LIN {X 62.948,Y 54.532,Z 81.721,A 180.000,B 0.000,C 180.000} C_DIS
LIN {X 62.927,Y 54.455,Z 81.718,A 180.000,B 0.000,C 180.000} C_DIS
LIN {X 62.907,Y 54.379,Z 81.716,A 180.000,B 0.000,C 180.000} C_DIS
LIN {X 62.887,Y 54.303,Z 81.713,A 180.000,B 0.000,C 180.000} C_DIS
LIN {X 62.867,Y 54.226,Z 81.710,A 180.000,B 0.000,C 180.000} C_DIS
LIN {X 62.847,Y 54.150,Z 81.707,A 180.000,B 0.000,C 180.000} C_DIS
LIN {X 62.806,Y 53.998,Z 81.702,A 180.000,B 0.000,C 180.000} C_DIS
LIN {X 62.746,Y 53.769,Z 81.693,A 180.000,B 0.000,C 180.000} C_DIS
LIN {X 62.706,Y 53.616,Z 81.688,A 180.000,B 0.000,C 180.000} C_DIS
LIN {X 62.686,Y 53.540,Z 81.685,A 180.000,B 0.000,C 180.000} C_DIS
LIN {X 62.645,Y 53.387,Z 81.680,A 180.000,B 0.000,C 180.000} C_DIS
LIN {X 62.585,Y 53.158,Z 81.671,A 180.000,B 0.000,C 180.000} C_DIS
LIN {X 62.544,Y 53.006,Z 81.666,A 180.000,B 0.000,C 180.000} C_DIS
LIN {X 62.524,Y 52.929,Z 81.663,A 180.000,B 0.000,C 180.000} C_DIS
LIN {X 62.484,Y 52.777,Z 81.658,A 180.000,B 0.000,C 180.000} C_DIS
LIN {X 62.423,Y 52.548,Z 81.649,A 180.000,B 0.000,C 180.000} C_DIS
LIN {X 62.383,Y 52.395,Z 81.644,A 180.000,B 0.000,C 180.000} C_DIS
LIN {X 62.363,Y 52.319,Z 81.641,A 180.000,B 0.000,C 180.000} C_DIS
LIN {X 62.323,Y 52.166,Z 81.636,A 180.000,B 0.000,C 180.000} C_DIS
LIN {X 62.262,Y 51.937,Z 81.627,A 180.000,B 0.000,C 180.000} C_DIS
LIN {X 62.222,Y 51.785,Z 81.622,A 180.000,B 0.000,C 180.000} C_DIS
LIN {X 62.202,Y 51.708,Z 81.619,A 180.000,B 0.000,C 180.000} C_DIS
LIN {X 62.161,Y 51.556,Z 81.614,A 180.000,B 0.000,C 180.000} C_DIS
LIN {X 62.040,Y 51.098,Z 81.597,A 180.000,B 0.000,C 180.000} C_DIS
LIN {X 62.000,Y 50.945,Z 81.592,A 180.000,B 0.000,C 180.000} C_DIS
LIN {X 61.939,Y 50.716,Z 81.583,A 180.000,B 0.000,C 180.000} C_DIS
LIN {X 61.816,Y 50.259,Z 81.567,A 180.000,B 0.000,C 180.000} C_DIS
LIN {X 61.775,Y 50.107,Z 81.561,A 180.000,B 0.000,C 180.000} C_DIS
LIN {X 61.651,Y 49.650,Z 81.545,A 180.000,B 0.000,C 180.000} C_DIS
LIN {X 61.568,Y 49.345,Z 81.534,A 180.000,B 0.000,C 180.000} C_DIS
LIN {X 61.465,Y 48.965,Z 81.520,A 180.000,B 0.000,C 180.000} C_DIS
LIN {X 61.218,Y 48.051,Z 81.487,A 180.000,B 0.000,C 180.000} C_DIS
LIN {X 61.099,Y 47.612,Z 81.471,A 180.000,B 0.000,C 180.000} C_DIS
LIN {X 61.062,Y 47.478,Z 81.466,A 180.000,B 0.000,C 180.000} C_DIS
LIN {X 61.028,Y 47.375,Z 81.462,A 180.000,B 0.000,C 180.000} C_DIS
LIN {X 60.990,Y 47.272,Z 81.458,A 180.000,B 0.000,C 180.000} C_DIS
LIN {X 60.946,Y 47.169,Z 81.455,A 180.000,B 0.000,C 180.000} C_DIS
LIN {X 60.897,Y 47.067,Z 81.451,A 180.000,B 0.000,C 180.000} C_DIS
LIN {X 60.844,Y 46.969,Z 81.447,A 180.000,B 0.000,C 180.000} C_DIS
LIN {X 60.787,Y 46.873,Z 81.443,A 180.000,B 0.000,C 180.000} C_DIS
LIN {X 60.719,Y 46.772,Z 81.439,A 180.000,B 0.000,C 180.000} C_DIS
LIN {X 60.646,Y 46.673,Z 81.434,A 180.000,B 0.000,C 180.000} C_DIS
LIN {X 60.566,Y 46.577,Z 81.430,A 180.000,B 0.000,C 180.000} C_DIS
LIN {X 60.482,Y 46.486,Z 81.426,A 180.000,B 0.000,C 180.000} C_DIS
LIN {X 60.397,Y 46.403,Z 81.421,A 180.000,B 0.000,C 180.000} C_DIS
LIN {X 60.308,Y 46.324,Z 81.417,A 180.000,B 0.000,C 180.000} C_DIS
LIN {X 60.206,Y 46.243,Z 81.413,A 180.000,B 0.000,C 180.000} C_DIS
LIN {X 60.099,Y 46.167,Z 81.408,A 180.000,B 0.000,C 180.000} C_DIS
LIN {X 59.980,Y 46.093,Z 81.403,A 180.000,B 0.000,C 180.000} C_DIS
LIN {X 59.857,Y 46.027,Z 81.398,A 180.000,B 0.000,C 180.000} C_DIS
LIN {X 59.733,Y 45.969,Z 81.394,A 180.000,B 0.000,C 180.000} C_DIS
LIN {X 59.605,Y 45.918,Z 81.389,A 180.000,B 0.000,C 180.000} C_DIS
LIN {X 59.537,Y 45.895,Z 81.386,A 180.000,B 0.000,C 180.000} C_DIS
LIN {X 59.467,Y 45.874,Z 81.384,A 180.000,B 0.000,C 180.000} C_DIS
LIN {X 59.397,Y 45.855,Z 81.381,A 180.000,B 0.000,C 180.000} C_DIS
LIN {X 59.327,Y 45.838,Z 81.379,A 180.000,B 0.000,C 180.000} C_DIS
LIN {X 59.253,Y 45.823,Z 81.376,A 180.000,B 0.000,C 180.000} C_DIS
LIN {X 59.179,Y 45.810,Z 81.373,A 180.000,B 0.000,C 180.000} C_DIS
LIN {X 59.104,Y 45.800,Z 81.371,A 180.000,B 0.000,C 180.000} C_DIS
LIN {X 59.029,Y 45.793,Z 81.368,A 180.000,B 0.000,C 180.000} C_DIS
LIN {X 58.952,Y 45.788,Z 81.366,A 180.000,B 0.000,C 180.000} C_DIS
LIN {X 58.874,Y 45.785,Z 81.363,A 180.000,B 0.000,C 180.000} C_DIS
LIN {X 58.797,Y 45.786,Z 81.360,A 180.000,B 0.000,C 180.000} C_DIS
LIN {X 58.720,Y 45.789,Z 81.357,A 180.000,B 0.000,C 180.000} C_DIS
LIN {X 58.640,Y 45.795,Z 81.355,A 180.000,B 0.000,C 180.000} C_DIS
LIN {X 58.560,Y 45.803,Z 81.352,A 180.000,B 0.000,C 180.000} C_DIS
LIN {X 58.481,Y 45.815,Z 81.349,A 180.000,B 0.000,C 180.000} C_DIS
LIN {X 58.402,Y 45.829,Z 81.346,A 180.000,B 0.000,C 180.000} C_DIS
LIN {X 58.325,Y 45.846,Z 81.343,A 180.000,B 0.000,C 180.000} C_DIS
LIN {X 58.248,Y 45.866,Z 81.341,A 180.000,B 0.000,C 180.000} C_DIS
LIN {X 58.173,Y 45.889,Z 81.338,A 180.000,B 0.000,C 180.000} C_DIS
LIN {X 58.098,Y 45.913,Z 81.335,A 180.000,B 0.000,C 180.000} C_DIS
LIN {X 57.949,Y 45.964,Z 81.330,A 180.000,B 0.000,C 180.000} C_DIS
LIN {X 57.501,Y 46.115,Z 81.313,A 180.000,B 0.000,C 180.000} C_DIS
LIN {X 57.352,Y 46.165,Z 81.308,A 180.000,B 0.000,C 180.000} C_DIS
LIN {X 56.904,Y 46.316,Z 81.291,A 180.000,B 0.000,C 180.000} C_DIS
LIN {X 56.755,Y 46.367,Z 81.286,A 180.000,B 0.000,C 180.000} C_DIS
LIN {X 56.531,Y 46.442,Z 81.277,A 180.000,B 0.000,C 180.000} C_DIS
LIN {X 56.382,Y 46.492,Z 81.272,A 180.000,B 0.000,C 180.000} C_DIS
LIN {X 56.307,Y 46.518,Z 81.269,A 180.000,B 0.000,C 180.000} C_DIS
LIN {X 56.158,Y 46.568,Z 81.264,A 180.000,B 0.000,C 180.000} C_DIS
LIN {X 55.934,Y 46.643,Z 81.255,A 180.000,B 0.000,C 180.000} C_DIS
LIN {X 55.785,Y 46.694,Z 81.250,A 180.000,B 0.000,C 180.000} C_DIS
LIN {X 55.710,Y 46.719,Z 81.247,A 180.000,B 0.000,C 180.000} C_DIS
LIN {X 55.561,Y 46.769,Z 81.242,A 180.000,B 0.000,C 180.000} C_DIS
LIN {X 55.337,Y 46.845,Z 81.233,A 180.000,B 0.000,C 180.000} C_DIS
LIN {X 55.188,Y 46.895,Z 81.228,A 180.000,B 0.000,C 180.000} C_DIS
LIN {X 55.113,Y 46.920,Z 81.225,A 180.000,B 0.000,C 180.000} C_DIS
LIN {X 54.964,Y 46.971,Z 81.220,A 180.000,B 0.000,C 180.000} C_DIS
LIN {X 54.740,Y 47.046,Z 81.211,A 180.000,B 0.000,C 180.000} C_DIS
LIN {X 54.591,Y 47.097,Z 81.206,A 180.000,B 0.000,C 180.000} C_DIS
LIN {X 54.516,Y 47.122,Z 81.203,A 180.000,B 0.000,C 180.000} C_DIS
LIN {X 54.367,Y 47.172,Z 81.198,A 180.000,B 0.000,C 180.000} C_DIS
LIN {X 54.143,Y 47.248,Z 81.189,A 180.000,B 0.000,C 180.000} C_DIS
LIN {X 53.994,Y 47.298,Z 81.184,A 180.000,B 0.000,C 180.000} C_DIS
LIN {X 53.845,Y 47.348,Z 81.179,A 180.000,B 0.000,C 180.000} C_DIS
LIN {X 53.695,Y 47.399,Z 81.173,A 180.000,B 0.000,C 180.000} C_DIS
LIN {X 53.546,Y 47.449,Z 81.168,A 180.000,B 0.000,C 180.000} C_DIS
LIN {X 53.397,Y 47.499,Z 81.163,A 180.000,B 0.000,C 180.000} C_DIS
LIN {X 53.322,Y 47.524,Z 81.160,A 180.000,B 0.000,C 180.000} C_DIS
LIN {X 53.248,Y 47.550,Z 81.158,A 180.000,B 0.000,C 180.000} C_DIS
LIN {X 53.173,Y 47.575,Z 81.155,A 180.000,B 0.000,C 180.000} C_DIS
LIN {X 53.098,Y 47.600,Z 81.153,A 180.000,B 0.000,C 180.000} C_DIS
LIN {X 53.024,Y 47.625,Z 81.150,A 180.000,B 0.000,C 180.000} C_DIS
LIN {X 52.949,Y 47.650,Z 81.147,A 180.000,B 0.000,C 180.000} C_DIS
LIN {X 52.875,Y 47.675,Z 81.145,A 180.000,B 0.000,C 180.000} C_DIS
LIN {X 52.725,Y 47.726,Z 81.140,A 180.000,B 0.000,C 180.000} C_DIS
LIN {X 52.576,Y 47.776,Z 81.135,A 180.000,B 0.000,C 180.000} C_DIS
LIN {X 52.427,Y 47.827,Z 81.130,A 180.000,B 0.000,C 180.000} C_DIS
LIN {X 52.278,Y 47.877,Z 81.126,A 180.000,B 0.000,C 180.000} C_DIS
LIN {X 52.128,Y 47.927,Z 81.121,A 180.000,B 0.000,C 180.000} C_DIS
LIN {X 51.979,Y 47.978,Z 81.116,A 180.000,B 0.000,C 180.000} C_DIS
LIN {X 51.830,Y 48.028,Z 81.112,A 180.000,B 0.000,C 180.000} C_DIS
LIN {X 51.681,Y 48.078,Z 81.107,A 180.000,B 0.000,C 180.000} C_DIS
LIN {X 51.531,Y 48.129,Z 81.103,A 180.000,B 0.000,C 180.000} C_DIS
LIN {X 51.382,Y 48.179,Z 81.099,A 180.000,B 0.000,C 180.000} C_DIS
LIN {X 51.233,Y 48.229,Z 81.094,A 180.000,B 0.000,C 180.000} C_DIS
LIN {X 51.084,Y 48.280,Z 81.090,A 180.000,B 0.000,C 180.000} C_DIS
LIN {X 50.935,Y 48.330,Z 81.086,A 180.000,B 0.000,C 180.000} C_DIS
LIN {X 50.785,Y 48.380,Z 81.082,A 180.000,B 0.000,C 180.000} C_DIS
LIN {X 50.636,Y 48.431,Z 81.078,A 180.000,B 0.000,C 180.000} C_DIS
LIN {X 50.487,Y 48.481,Z 81.074,A 180.000,B 0.000,C 180.000} C_DIS
LIN {X 50.338,Y 48.531,Z 81.071,A 180.000,B 0.000,C 180.000} C_DIS
LIN {X 50.188,Y 48.582,Z 81.067,A 180.000,B 0.000,C 180.000} C_DIS
LIN {X 50.039,Y 48.632,Z 81.063,A 180.000,B 0.000,C 180.000} C_DIS
LIN {X 49.890,Y 48.682,Z 81.060,A 180.000,B 0.000,C 180.000} C_DIS
LIN {X 49.741,Y 48.733,Z 81.057,A 180.000,B 0.000,C 180.000} C_DIS
LIN {X 49.591,Y 48.783,Z 81.053,A 180.000,B 0.000,C 180.000} C_DIS
LIN {X 49.442,Y 48.833,Z 81.050,A 180.000,B 0.000,C 180.000} C_DIS
LIN {X 49.293,Y 48.884,Z 81.047,A 180.000,B 0.000,C 180.000} C_DIS
LIN {X 49.144,Y 48.934,Z 81.044,A 180.000,B 0.000,C 180.000} C_DIS
LIN {X 48.994,Y 48.984,Z 81.041,A 180.000,B 0.000,C 180.000} C_DIS
LIN {X 48.845,Y 49.035,Z 81.038,A 180.000,B 0.000,C 180.000} C_DIS
LIN {X 48.696,Y 49.085,Z 81.035,A 180.000,B 0.000,C 180.000} C_DIS
LIN {X 48.547,Y 49.135,Z 81.032,A 180.000,B 0.000,C 180.000} C_DIS
LIN {X 48.398,Y 49.186,Z 81.030,A 180.000,B 0.000,C 180.000} C_DIS
LIN {X 48.248,Y 49.236,Z 81.027,A 180.000,B 0.000,C 180.000} C_DIS
LIN {X 47.950,Y 49.337,Z 81.023,A 180.000,B 0.000,C 180.000} C_DIS
LIN {X 47.651,Y 49.438,Z 81.019,A 180.000,B 0.000,C 180.000} C_DIS
LIN {X 47.353,Y 49.538,Z 81.015,A 180.000,B 0.000,C 180.000} C_DIS
LIN {X 47.054,Y 49.639,Z 81.011,A 180.000,B 0.000,C 180.000} C_DIS
LIN {X 46.756,Y 49.740,Z 81.008,A 180.000,B 0.000,C 180.000} C_DIS
LIN {X 46.457,Y 49.840,Z 81.006,A 180.000,B 0.000,C 180.000} C_DIS
LIN {X 46.159,Y 49.941,Z 81.004,A 180.000,B 0.000,C 180.000} C_DIS
LIN {X 46.085,Y 49.969,Z 81.003,A 180.000,B 0.000,C 180.000} C_DIS
LIN {X 46.013,Y 49.999,Z 81.003,A 180.000,B 0.000,C 180.000} C_DIS
LIN {X 45.941,Y 50.032,Z 81.002,A 180.000,B 0.000,C 180.000} C_DIS
LIN {X 45.870,Y 50.066,Z 81.002,A 180.000,B 0.000,C 180.000} C_DIS
LIN {X 45.800,Y 50.103,Z 81.002,A 180.000,B 0.000,C 180.000} C_DIS
LIN {X 45.732,Y 50.142,Z 81.001,A 180.000,B 0.000,C 180.000} C_DIS
LIN {X 45.665,Y 50.183,Z 81.001,A 180.000,B 0.000,C 180.000} C_DIS
LIN {X 45.599,Y 50.226,Z 81.001,A 180.000,B 0.000,C 180.000} C_DIS
LIN {X 45.534,Y 50.271,Z 81.001,A 180.000,B 0.000,C 180.000} C_DIS
LIN {X 45.471,Y 50.318,Z 81.000,A 180.000,B 0.000,C 180.000} C_DIS
LIN {X 45.410,Y 50.367,Z 81.000,A 180.000,B 0.000,C 180.000} C_DIS
LIN {X 45.350,Y 50.418,Z 81.000,A 180.000,B 0.000,C 180.000} C_DIS
LIN {X 45.250,Y 50.511,Z 81.000,A 180.000,B 0.000,C 180.000} C_DIS
LIN {X 45.156,Y 50.609,Z 81.000,A 180.000,B 0.000,C 180.000} C_DIS
; Cutting Move Starts
LIN {X 45.053,Y 50.728,Z 81.000,A 180.000,B 0.000,C 180.000} C_DIS
LIN {X 45.017,Y 50.774,Z 81.000,A 180.000,B 0.000,C 180.000} C_DIS
LIN {X 44.952,Y 50.863,Z 81.000,A 180.000,B 0.000,C 180.000} C_DIS
LIN {X 44.892,Y 50.953,Z 81.000,A 180.000,B 0.000,C 180.000} C_DIS
LIN {X 44.874,Y 50.981,Z 81.000,A 180.000,B 0.000,C 180.000} C_DIS
LIN {X 44.788,Y 51.131,Z 81.000,A 180.000,B 0.000,C 180.000} C_DIS
LIN {X 44.703,Y 51.310,Z 81.000,A 180.000,B 0.000,C 180.000} C_DIS
LIN {X 44.696,Y 51.328,Z 81.000,A 180.000,B 0.000,C 180.000} C_DIS
LIN {X 44.634,Y 51.489,Z 81.000,A 180.000,B 0.000,C 180.000} C_DIS
LIN {X 44.581,Y 51.668,Z 81.000,A 180.000,B 0.000,C 180.000} C_DIS
LIN {X 44.541,Y 51.847,Z 81.000,A 180.000,B 0.000,C 180.000} C_DIS
LIN {X 44.517,Y 52.012,Z 81.000,A 180.000,B 0.000,C 180.000} C_DIS
LIN {X 44.515,Y 52.025,Z 81.000,A 180.000,B 0.000,C 180.000} C_DIS
LIN {X 44.503,Y 52.204,Z 81.000,A 180.000,B 0.000,C 180.000} C_DIS
LIN {X 44.502,Y 52.383,Z 81.000,A 180.000,B 0.000,C 180.000} C_DIS
LIN {X 44.515,Y 52.562,Z 81.000,A 180.000,B 0.000,C 180.000} C_DIS
LIN {X 44.517,Y 52.579,Z 81.000,A 180.000,B 0.000,C 180.000} C_DIS
LIN {X 44.541,Y 52.740,Z 81.000,A 180.000,B 0.000,C 180.000} C_DIS
LIN {X 44.580,Y 52.919,Z 81.000,A 180.000,B 0.000,C 180.000} C_DIS
LIN {X 44.633,Y 53.098,Z 81.000,A 180.000,B 0.000,C 180.000} C_DIS
LIN {X 51.026,Y 72.048,Z 81.000,A 180.000,B 0.000,C 180.000} C_DIS
LIN {X 51.094,Y 72.226,Z 81.000,A 180.000,B 0.000,C 180.000} C_DIS
LIN {X 51.131,Y 72.310,Z 81.000,A 180.000,B 0.000,C 180.000} C_DIS
LIN {X 51.179,Y 72.405,Z 81.000,A 180.000,B 0.000,C 180.000} C_DIS
LIN {X 51.282,Y 72.584,Z 81.000,A 180.000,B 0.000,C 180.000} C_DIS
LIN {X 51.310,Y 72.628,Z 81.000,A 180.000,B 0.000,C 180.000} C_DIS
LIN {X 51.406,Y 72.763,Z 81.000,A 180.000,B 0.000,C 180.000} C_DIS
LIN {X 51.489,Y 72.865,Z 81.000,A 180.000,B 0.000,C 180.000} C_DIS
LIN {X 51.556,Y 72.941,Z 81.000,A 180.000,B 0.000,C 180.000} C_DIS
LIN {X 51.668,Y 73.055,Z 81.000,A 180.000,B 0.000,C 180.000} C_DIS
LIN {X 51.739,Y 73.120,Z 81.000,A 180.000,B 0.000,C 180.000} C_DIS
LIN {X 51.847,Y 73.210,Z 81.000,A 180.000,B 0.000,C 180.000} C_DIS
LIN {X 51.967,Y 73.299,Z 81.000,A 180.000,B 0.000,C 180.000} C_DIS
LIN {X 52.025,Y 73.338,Z 81.000,A 180.000,B 0.000,C 180.000} C_DIS
LIN {X 52.204,Y 73.445,Z 81.000,A 180.000,B 0.000,C 180.000} C_DIS
LIN {X 52.267,Y 73.478,Z 81.000,A 180.000,B 0.000,C 180.000} C_DIS
LIN {X 52.383,Y 73.533,Z 81.000,A 180.000,B 0.000,C 180.000} C_DIS
LIN {X 52.562,Y 73.604,Z 81.000,A 180.000,B 0.000,C 180.000} C_DIS
LIN {X 52.730,Y 73.656,Z 81.000,A 180.000,B 0.000,C 180.000} C_DIS
LIN {X 52.740,Y 73.659,Z 81.000,A 180.000,B 0.000,C 180.000} C_DIS
LIN {X 52.919,Y 73.701,Z 81.000,A 180.000,B 0.000,C 180.000} C_DIS
LIN {X 53.009,Y 73.716,Z 81.000,A 180.000,B 0.000,C 180.000} C_DIS
LIN {X 53.098,Y 73.729,Z 81.000,A 180.000,B 0.000,C 180.000} C_DIS
LIN {X 53.187,Y 73.738,Z 81.000,A 180.000,B 0.000,C 180.000} C_DIS
LIN {X 53.277,Y 73.743,Z 81.000,A 180.000,B 0.000,C 180.000} C_DIS
LIN {X 53.366,Y 73.746,Z 81.000,A 180.000,B 0.000,C 180.000} C_DIS
LIN {X 53.455,Y 73.745,Z 81.000,A 180.000,B 0.000,C 180.000} C_DIS
LIN {X 53.545,Y 73.742,Z 81.000,A 180.000,B 0.000,C 180.000} C_DIS
LIN {X 53.634,Y 73.735,Z 81.000,A 180.000,B 0.000,C 180.000} C_DIS
LIN {X 53.724,Y 73.724,Z 81.000,A 180.000,B 0.000,C 180.000} C_DIS
LIN {X 53.813,Y 73.711,Z 81.000,A 180.000,B 0.000,C 180.000} C_DIS
LIN {X 53.902,Y 73.694,Z 81.000,A 180.000,B 0.000,C 180.000} C_DIS
LIN {X 53.992,Y 73.674,Z 81.000,A 180.000,B 0.000,C 180.000} C_DIS
LIN {X 54.057,Y 73.656,Z 81.000,A 180.000,B 0.000,C 180.000} C_DIS
LIN {X 54.171,Y 73.622,Z 81.000,A 180.000,B 0.000,C 180.000} C_DIS
LIN {X 54.349,Y 73.562,Z 81.000,A 180.000,B 0.000,C 180.000} C_DIS
LIN {X 66.506,Y 69.461,Z 81.000,A 180.000,B 0.000,C 180.000} C_DIS
LIN {X 66.684,Y 69.401,Z 81.000,A 180.000,B 0.000,C 180.000} C_DIS
LIN {X 66.777,Y 69.366,Z 81.000,A 180.000,B 0.000,C 180.000} C_DIS
LIN {X 66.863,Y 69.330,Z 81.000,A 180.000,B 0.000,C 180.000} C_DIS
LIN {X 66.953,Y 69.288,Z 81.000,A 180.000,B 0.000,C 180.000} C_DIS
LIN {X 67.042,Y 69.242,Z 81.000,A 180.000,B 0.000,C 180.000} C_DIS
LIN {X 67.137,Y 69.187,Z 81.000,A 180.000,B 0.000,C 180.000} C_DIS
LIN {X 67.221,Y 69.135,Z 81.000,A 180.000,B 0.000,C 180.000} C_DIS
LIN {X 67.309,Y 69.074,Z 81.000,A 180.000,B 0.000,C 180.000} C_DIS
LIN {X 67.396,Y 69.008,Z 81.000,A 180.000,B 0.000,C 180.000} C_DIS
LIN {X 67.399,Y 69.006,Z 81.000,A 180.000,B 0.000,C 180.000} C_DIS
LIN {X 67.489,Y 68.932,Z 81.000,A 180.000,B 0.000,C 180.000} C_DIS
LIN {X 67.578,Y 68.850,Z 81.000,A 180.000,B 0.000,C 180.000} C_DIS
LIN {X 67.600,Y 68.830,Z 81.000,A 180.000,B 0.000,C 180.000} C_DIS
LIN {X 67.682,Y 68.745,Z 81.000,A 180.000,B 0.000,C 180.000} C_DIS
LIN {X 67.757,Y 68.661,Z 81.000,A 180.000,B 0.000,C 180.000} C_DIS
LIN {X 67.765,Y 68.651,Z 81.000,A 180.000,B 0.000,C 180.000} C_DIS
LIN {X 67.837,Y 68.562,Z 81.000,A 180.000,B 0.000,C 180.000} C_DIS
LIN {X 67.902,Y 68.472,Z 81.000,A 180.000,B 0.000,C 180.000} C_DIS
LIN {X 67.936,Y 68.422,Z 81.000,A 180.000,B 0.000,C 180.000} C_DIS
LIN {X 68.015,Y 68.293,Z 81.000,A 180.000,B 0.000,C 180.000} C_DIS
LIN {X 68.109,Y 68.115,Z 81.000,A 180.000,B 0.000,C 180.000} C_DIS
LIN {X 68.115,Y 68.103,Z 81.000,A 180.000,B 0.000,C 180.000} C_DIS
LIN {X 68.186,Y 67.936,Z 81.000,A 180.000,B 0.000,C 180.000} C_DIS
LIN {X 68.246,Y 67.757,Z 81.000,A 180.000,B 0.000,C 180.000} C_DIS
LIN {X 68.292,Y 67.578,Z 81.000,A 180.000,B 0.000,C 180.000} C_DIS
LIN {X 68.293,Y 67.573,Z 81.000,A 180.000,B 0.000,C 180.000} C_DIS
LIN {X 68.325,Y 67.399,Z 81.000,A 180.000,B 0.000,C 180.000} C_DIS
LIN {X 68.344,Y 67.221,Z 81.000,A 180.000,B 0.000,C 180.000} C_DIS
LIN {X 68.350,Y 67.042,Z 81.000,A 180.000,B 0.000,C 180.000} C_DIS
LIN {X 68.343,Y 66.863,Z 81.000,A 180.000,B 0.000,C 180.000} C_DIS
LIN {X 68.324,Y 66.684,Z 81.000,A 180.000,B 0.000,C 180.000} C_DIS
LIN {X 68.293,Y 66.515,Z 81.000,A 180.000,B 0.000,C 180.000} C_DIS
LIN {X 68.291,Y 66.506,Z 81.000,A 180.000,B 0.000,C 180.000} C_DIS
LIN {X 68.245,Y 66.327,Z 81.000,A 180.000,B 0.000,C 180.000} C_DIS
LIN {X 68.186,Y 66.148,Z 81.000,A 180.000,B 0.000,C 180.000} C_DIS
LIN {X 61.854,Y 47.377,Z 81.000,A 180.000,B 0.000,C 180.000} C_DIS
LIN {X 61.791,Y 47.198,Z 81.000,A 180.000,B 0.000,C 180.000} C_DIS
LIN {X 61.715,Y 47.020,Z 81.000,A 180.000,B 0.000,C 180.000} C_DIS
LIN {X 61.679,Y 46.947,Z 81.000,A 180.000,B 0.000,C 180.000} C_DIS
LIN {X 61.621,Y 46.841,Z 81.000,A 180.000,B 0.000,C 180.000} C_DIS
LIN {X 61.507,Y 46.662,Z 81.000,A 180.000,B 0.000,C 180.000} C_DIS
LIN {X 61.500,Y 46.653,Z 81.000,A 180.000,B 0.000,C 180.000} C_DIS
LIN {X 61.370,Y 46.483,Z 81.000,A 180.000,B 0.000,C 180.000} C_DIS
LIN {X 61.321,Y 46.428,Z 81.000,A 180.000,B 0.000,C 180.000} C_DIS
LIN {X 61.204,Y 46.305,Z 81.000,A 180.000,B 0.000,C 180.000} C_DIS
LIN {X 61.143,Y 46.247,Z 81.000,A 180.000,B 0.000,C 180.000} C_DIS
LIN {X 60.999,Y 46.126,Z 81.000,A 180.000,B 0.000,C 180.000} C_DIS
LIN {X 60.964,Y 46.098,Z 81.000,A 180.000,B 0.000,C 180.000} C_DIS
LIN {X 60.785,Y 45.975,Z 81.000,A 180.000,B 0.000,C 180.000} C_DIS
LIN {X 60.739,Y 45.947,Z 81.000,A 180.000,B 0.000,C 180.000} C_DIS
LIN {X 60.606,Y 45.873,Z 81.000,A 180.000,B 0.000,C 180.000} C_DIS
LIN {X 60.427,Y 45.789,Z 81.000,A 180.000,B 0.000,C 180.000} C_DIS
LIN {X 60.376,Y 45.768,Z 81.000,A 180.000,B 0.000,C 180.000} C_DIS
LIN {X 60.249,Y 45.722,Z 81.000,A 180.000,B 0.000,C 180.000} C_DIS
LIN {X 60.070,Y 45.670,Z 81.000,A 180.000,B 0.000,C 180.000} C_DIS
LIN {X 59.891,Y 45.631,Z 81.000,A 180.000,B 0.000,C 180.000} C_DIS
LIN {X 59.802,Y 45.617,Z 81.000,A 180.000,B 0.000,C 180.000} C_DIS
LIN {X 59.712,Y 45.606,Z 81.000,A 180.000,B 0.000,C 180.000} C_DIS
LIN {X 59.623,Y 45.599,Z 81.000,A 180.000,B 0.000,C 180.000} C_DIS
LIN {X 59.534,Y 45.595,Z 81.000,A 180.000,B 0.000,C 180.000} C_DIS
LIN {X 59.444,Y 45.593,Z 81.000,A 180.000,B 0.000,C 180.000} C_DIS
LIN {X 59.355,Y 45.595,Z 81.000,A 180.000,B 0.000,C 180.000} C_DIS
LIN {X 59.265,Y 45.601,Z 81.000,A 180.000,B 0.000,C 180.000} C_DIS
LIN {X 59.176,Y 45.609,Z 81.000,A 180.000,B 0.000,C 180.000} C_DIS
LIN {X 59.087,Y 45.621,Z 81.000,A 180.000,B 0.000,C 180.000} C_DIS
LIN {X 58.997,Y 45.636,Z 81.000,A 180.000,B 0.000,C 180.000} C_DIS
LIN {X 58.908,Y 45.654,Z 81.000,A 180.000,B 0.000,C 180.000} C_DIS
LIN {X 58.819,Y 45.676,Z 81.000,A 180.000,B 0.000,C 180.000} C_DIS
LIN {X 58.729,Y 45.702,Z 81.000,A 180.000,B 0.000,C 180.000} C_DIS
LIN {X 58.640,Y 45.731,Z 81.000,A 180.000,B 0.000,C 180.000} C_DIS
LIN {X 46.305,Y 49.892,Z 81.000,A 180.000,B 0.000,C 180.000} C_DIS
LIN {X 46.126,Y 49.954,Z 81.000,A 180.000,B 0.000,C 180.000} C_DIS
LIN {X 46.036,Y 49.989,Z 81.000,A 180.000,B 0.000,C 180.000} C_DIS
LIN {X 45.947,Y 50.028,Z 81.000,A 180.000,B 0.000,C 180.000} C_DIS
LIN {X 45.884,Y 50.059,Z 81.000,A 180.000,B 0.000,C 180.000} C_DIS
LIN {X 45.826,Y 50.089,Z 81.000,A 180.000,B 0.000,C 180.000} C_DIS
LIN {X 45.768,Y 50.120,Z 81.000,A 180.000,B 0.000,C 180.000} C_DIS
LIN {X 45.679,Y 50.173,Z 81.000,A 180.000,B 0.000,C 180.000} C_DIS
LIN {X 45.590,Y 50.232,Z 81.000,A 180.000,B 0.000,C 180.000} C_DIS
LIN {X 45.581,Y 50.238,Z 81.000,A 180.000,B 0.000,C 180.000} C_DIS
LIN {X 45.496,Y 50.299,Z 81.000,A 180.000,B 0.000,C 180.000} C_DIS
LIN {X 45.411,Y 50.366,Z 81.000,A 180.000,B 0.000,C 180.000} C_DIS
LIN {X 45.352,Y 50.416,Z 81.000,A 180.000,B 0.000,C 180.000} C_DIS
LIN {X 45.232,Y 50.529,Z 81.000,A 180.000,B 0.000,C 180.000} C_DIS
LIN {X 45.168,Y 50.595,Z 81.000,A 180.000,B 0.000,C 180.000} C_DIS
LIN {X 45.156,Y 50.609,Z 81.000,A 180.000,B 0.000,C 180.000} C_DIS
; Link Move Starts
LIN {X 45.061,Y 50.718,Z 81.000,A 180.000,B 0.000,C 180.000} C_DIS
LIN {X 44.974,Y 50.832,Z 81.000,A 180.000,B 0.000,C 180.000} C_DIS
LIN {X 44.894,Y 50.948,Z 81.000,A 180.000,B 0.000,C 180.000} C_DIS
LIN {X 44.822,Y 51.068,Z 80.999,A 180.000,B 0.000,C 180.000} C_DIS
LIN {X 44.761,Y 51.182,Z 80.999,A 180.000,B 0.000,C 180.000} C_DIS
LIN {X 44.706,Y 51.299,Z 80.998,A 180.000,B 0.000,C 180.000} C_DIS
LIN {X 44.657,Y 51.418,Z 80.998,A 180.000,B 0.000,C 180.000} C_DIS
LIN {X 44.614,Y 51.539,Z 80.997,A 180.000,B 0.000,C 180.000} C_DIS
LIN {X 44.553,Y 51.760,Z 80.996,A 180.000,B 0.000,C 180.000} C_DIS
LIN {X 44.527,Y 51.892,Z 80.995,A 180.000,B 0.000,C 180.000} C_DIS
LIN {X 44.507,Y 52.025,Z 80.994,A 180.000,B 0.000,C 180.000} C_DIS
LIN {X 44.490,Y 52.238,Z 80.992,A 180.000,B 0.000,C 180.000} C_DIS
LIN {X 44.491,Y 52.450,Z 80.990,A 180.000,B 0.000,C 180.000} C_DIS
LIN {X 44.512,Y 52.682,Z 80.988,A 180.000,B 0.000,C 180.000} C_DIS
LIN {X 44.531,Y 52.799,Z 80.986,A 180.000,B 0.000,C 180.000} C_DIS
LIN {X 44.555,Y 52.914,Z 80.985,A 180.000,B 0.000,C 180.000} C_DIS
LIN {X 44.611,Y 53.117,Z 80.983,A 180.000,B 0.000,C 180.000} C_DIS
LIN {X 44.705,Y 53.413,Z 80.978,A 180.000,B 0.000,C 180.000} C_DIS
LIN {X 44.799,Y 53.714,Z 80.974,A 180.000,B 0.000,C 180.000} C_DIS
LIN {X 44.892,Y 54.014,Z 80.969,A 180.000,B 0.000,C 180.000} C_DIS
LIN {X 44.939,Y 54.165,Z 80.966,A 180.000,B 0.000,C 180.000} C_DIS
LIN {X 44.985,Y 54.316,Z 80.964,A 180.000,B 0.000,C 180.000} C_DIS
LIN {X 45.031,Y 54.466,Z 80.961,A 180.000,B 0.000,C 180.000} C_DIS
LIN {X 45.078,Y 54.617,Z 80.958,A 180.000,B 0.000,C 180.000} C_DIS
LIN {X 45.124,Y 54.768,Z 80.955,A 180.000,B 0.000,C 180.000} C_DIS
LIN {X 45.169,Y 54.918,Z 80.952,A 180.000,B 0.000,C 180.000} C_DIS
LIN {X 45.215,Y 55.069,Z 80.949,A 180.000,B 0.000,C 180.000} C_DIS
LIN {X 45.261,Y 55.220,Z 80.945,A 180.000,B 0.000,C 180.000} C_DIS
LIN {X 45.306,Y 55.371,Z 80.942,A 180.000,B 0.000,C 180.000} C_DIS
LIN {X 45.352,Y 55.522,Z 80.939,A 180.000,B 0.000,C 180.000} C_DIS
LIN {X 45.397,Y 55.673,Z 80.935,A 180.000,B 0.000,C 180.000} C_DIS
LIN {X 45.442,Y 55.824,Z 80.931,A 180.000,B 0.000,C 180.000} C_DIS
LIN {X 45.487,Y 55.975,Z 80.928,A 180.000,B 0.000,C 180.000} C_DIS
LIN {X 45.532,Y 56.126,Z 80.924,A 180.000,B 0.000,C 180.000} C_DIS
LIN {X 45.576,Y 56.277,Z 80.920,A 180.000,B 0.000,C 180.000} C_DIS
LIN {X 45.621,Y 56.428,Z 80.916,A 180.000,B 0.000,C 180.000} C_DIS
LIN {X 45.666,Y 56.579,Z 80.912,A 180.000,B 0.000,C 180.000} C_DIS
LIN {X 45.710,Y 56.731,Z 80.908,A 180.000,B 0.000,C 180.000} C_DIS
LIN {X 45.754,Y 56.882,Z 80.904,A 180.000,B 0.000,C 180.000} C_DIS
LIN {X 45.798,Y 57.033,Z 80.899,A 180.000,B 0.000,C 180.000} C_DIS
LIN {X 45.842,Y 57.185,Z 80.895,A 180.000,B 0.000,C 180.000} C_DIS
LIN {X 45.886,Y 57.336,Z 80.891,A 180.000,B 0.000,C 180.000} C_DIS
LIN {X 45.930,Y 57.487,Z 80.886,A 180.000,B 0.000,C 180.000} C_DIS
LIN {X 45.974,Y 57.639,Z 80.882,A 180.000,B 0.000,C 180.000} C_DIS
LIN {X 46.018,Y 57.790,Z 80.877,A 180.000,B 0.000,C 180.000} C_DIS
LIN {X 46.061,Y 57.942,Z 80.872,A 180.000,B 0.000,C 180.000} C_DIS
LIN {X 46.105,Y 58.093,Z 80.868,A 180.000,B 0.000,C 180.000} C_DIS
LIN {X 46.148,Y 58.245,Z 80.863,A 180.000,B 0.000,C 180.000} C_DIS
LIN {X 46.191,Y 58.397,Z 80.858,A 180.000,B 0.000,C 180.000} C_DIS
LIN {X 46.234,Y 58.548,Z 80.853,A 180.000,B 0.000,C 180.000} C_DIS
LIN {X 46.256,Y 58.624,Z 80.850,A 180.000,B 0.000,C 180.000} C_DIS
LIN {X 46.277,Y 58.700,Z 80.848,A 180.000,B 0.000,C 180.000} C_DIS
LIN {X 46.299,Y 58.776,Z 80.845,A 180.000,B 0.000,C 180.000} C_DIS
LIN {X 46.320,Y 58.852,Z 80.843,A 180.000,B 0.000,C 180.000} C_DIS
LIN {X 46.342,Y 58.928,Z 80.840,A 180.000,B 0.000,C 180.000} C_DIS
LIN {X 46.363,Y 59.004,Z 80.838,A 180.000,B 0.000,C 180.000} C_DIS
LIN {X 46.385,Y 59.079,Z 80.835,A 180.000,B 0.000,C 180.000} C_DIS
LIN {X 46.406,Y 59.155,Z 80.832,A 180.000,B 0.000,C 180.000} C_DIS
LIN {X 46.427,Y 59.231,Z 80.830,A 180.000,B 0.000,C 180.000} C_DIS
LIN {X 46.449,Y 59.307,Z 80.827,A 180.000,B 0.000,C 180.000} C_DIS
LIN {X 46.470,Y 59.383,Z 80.824,A 180.000,B 0.000,C 180.000} C_DIS
LIN {X 46.491,Y 59.459,Z 80.822,A 180.000,B 0.000,C 180.000} C_DIS
LIN {X 46.513,Y 59.535,Z 80.819,A 180.000,B 0.000,C 180.000} C_DIS
LIN {X 46.534,Y 59.611,Z 80.816,A 180.000,B 0.000,C 180.000} C_DIS
LIN {X 46.555,Y 59.687,Z 80.814,A 180.000,B 0.000,C 180.000} C_DIS
LIN {X 46.597,Y 59.839,Z 80.808,A 180.000,B 0.000,C 180.000} C_DIS
LIN {X 46.619,Y 59.915,Z 80.805,A 180.000,B 0.000,C 180.000} C_DIS
LIN {X 46.640,Y 59.991,Z 80.803,A 180.000,B 0.000,C 180.000} C_DIS
LIN {X 46.661,Y 60.067,Z 80.800,A 180.000,B 0.000,C 180.000} C_DIS
LIN {X 46.682,Y 60.143,Z 80.797,A 180.000,B 0.000,C 180.000} C_DIS
LIN {X 46.703,Y 60.219,Z 80.794,A 180.000,B 0.000,C 180.000} C_DIS
LIN {X 46.725,Y 60.295,Z 80.792,A 180.000,B 0.000,C 180.000} C_DIS
LIN {X 46.746,Y 60.370,Z 80.789,A 180.000,B 0.000,C 180.000} C_DIS
LIN {X 46.767,Y 60.446,Z 80.786,A 180.000,B 0.000,C 180.000} C_DIS
LIN {X 46.788,Y 60.522,Z 80.783,A 180.000,B 0.000,C 180.000} C_DIS
LIN {X 46.809,Y 60.598,Z 80.781,A 180.000,B 0.000,C 180.000} C_DIS
LIN {X 46.830,Y 60.674,Z 80.778,A 180.000,B 0.000,C 180.000} C_DIS
LIN {X 46.852,Y 60.750,Z 80.775,A 180.000,B 0.000,C 180.000} C_DIS
LIN {X 46.873,Y 60.826,Z 80.772,A 180.000,B 0.000,C 180.000} C_DIS
LIN {X 46.894,Y 60.902,Z 80.770,A 180.000,B 0.000,C 180.000} C_DIS
LIN {X 46.915,Y 60.978,Z 80.767,A 180.000,B 0.000,C 180.000} C_DIS
LIN {X 46.936,Y 61.054,Z 80.764,A 180.000,B 0.000,C 180.000} C_DIS
LIN {X 46.958,Y 61.130,Z 80.761,A 180.000,B 0.000,C 180.000} C_DIS
LIN {X 46.979,Y 61.206,Z 80.759,A 180.000,B 0.000,C 180.000} C_DIS
LIN {X 47.000,Y 61.282,Z 80.756,A 180.000,B 0.000,C 180.000} C_DIS
LIN {X 47.021,Y 61.358,Z 80.753,A 180.000,B 0.000,C 180.000} C_DIS
LIN {X 47.042,Y 61.434,Z 80.750,A 180.000,B 0.000,C 180.000} C_DIS
LIN {X 47.063,Y 61.510,Z 80.748,A 180.000,B 0.000,C 180.000} C_DIS
LIN {X 47.085,Y 61.586,Z 80.745,A 180.000,B 0.000,C 180.000} C_DIS
LIN {X 47.106,Y 61.662,Z 80.742,A 180.000,B 0.000,C 180.000} C_DIS
LIN {X 47.149,Y 61.814,Z 80.737,A 180.000,B 0.000,C 180.000} C_DIS
LIN {X 47.170,Y 61.890,Z 80.734,A 180.000,B 0.000,C 180.000} C_DIS
LIN {X 47.213,Y 62.041,Z 80.728,A 180.000,B 0.000,C 180.000} C_DIS
LIN {X 47.277,Y 62.269,Z 80.720,A 180.000,B 0.000,C 180.000} C_DIS
LIN {X 47.320,Y 62.421,Z 80.714,A 180.000,B 0.000,C 180.000} C_DIS
LIN {X 47.341,Y 62.497,Z 80.712,A 180.000,B 0.000,C 180.000} C_DIS
LIN {X 47.384,Y 62.648,Z 80.706,A 180.000,B 0.000,C 180.000} C_DIS
LIN {X 47.448,Y 62.876,Z 80.698,A 180.000,B 0.000,C 180.000} C_DIS
LIN {X 47.491,Y 63.028,Z 80.692,A 180.000,B 0.000,C 180.000} C_DIS
LIN {X 47.512,Y 63.104,Z 80.690,A 180.000,B 0.000,C 180.000} C_DIS
LIN {X 47.555,Y 63.256,Z 80.684,A 180.000,B 0.000,C 180.000} C_DIS
LIN {X 47.619,Y 63.483,Z 80.676,A 180.000,B 0.000,C 180.000} C_DIS
LIN {X 47.662,Y 63.635,Z 80.670,A 180.000,B 0.000,C 180.000} C_DIS
LIN {X 47.683,Y 63.711,Z 80.668,A 180.000,B 0.000,C 180.000} C_DIS
LIN {X 47.726,Y 63.863,Z 80.662,A 180.000,B 0.000,C 180.000} C_DIS
LIN {X 47.790,Y 64.091,Z 80.654,A 180.000,B 0.000,C 180.000} C_DIS
LIN {X 47.833,Y 64.242,Z 80.648,A 180.000,B 0.000,C 180.000} C_DIS
LIN {X 47.854,Y 64.318,Z 80.646,A 180.000,B 0.000,C 180.000} C_DIS
LIN {X 47.897,Y 64.470,Z 80.640,A 180.000,B 0.000,C 180.000} C_DIS
LIN {X 48.025,Y 64.925,Z 80.624,A 180.000,B 0.000,C 180.000} C_DIS
LIN {X 48.068,Y 65.077,Z 80.618,A 180.000,B 0.000,C 180.000} C_DIS
LIN {X 48.196,Y 65.533,Z 80.602,A 180.000,B 0.000,C 180.000} C_DIS
LIN {X 48.261,Y 65.760,Z 80.593,A 180.000,B 0.000,C 180.000} C_DIS
LIN {X 48.303,Y 65.912,Z 80.588,A 180.000,B 0.000,C 180.000} C_DIS
LIN {X 48.432,Y 66.367,Z 80.571,A 180.000,B 0.000,C 180.000} C_DIS
LIN {X 48.474,Y 66.519,Z 80.566,A 180.000,B 0.000,C 180.000} C_DIS
LIN {X 48.667,Y 67.202,Z 80.541,A 180.000,B 0.000,C 180.000} C_DIS
LIN {X 49.052,Y 68.568,Z 80.491,A 180.000,B 0.000,C 180.000} C_DIS
LIN {X 49.243,Y 69.247,Z 80.467,A 180.000,B 0.000,C 180.000} C_DIS
LIN {X 49.244,Y 69.251,Z 80.467,A 180.000,B 0.000,C 180.000} C_DIS
LIN {X 49.949,Y 71.341,Z 80.390,A 180.000,B 0.000,C 180.000} C_DIS
LIN {X 50.100,Y 71.788,Z 80.373,A 180.000,B 0.000,C 180.000} C_DIS
LIN {X 50.151,Y 71.938,Z 80.368,A 180.000,B 0.000,C 180.000} C_DIS
LIN {X 50.251,Y 72.236,Z 80.357,A 180.000,B 0.000,C 180.000} C_DIS
LIN {X 50.276,Y 72.311,Z 80.354,A 180.000,B 0.000,C 180.000} C_DIS
LIN {X 50.303,Y 72.385,Z 80.351,A 180.000,B 0.000,C 180.000} C_DIS
LIN {X 50.332,Y 72.458,Z 80.348,A 180.000,B 0.000,C 180.000} C_DIS
LIN {X 50.364,Y 72.530,Z 80.346,A 180.000,B 0.000,C 180.000} C_DIS
LIN {X 50.397,Y 72.602,Z 80.343,A 180.000,B 0.000,C 180.000} C_DIS
LIN {X 50.433,Y 72.672,Z 80.340,A 180.000,B 0.000,C 180.000} C_DIS
LIN {X 50.471,Y 72.741,Z 80.337,A 180.000,B 0.000,C 180.000} C_DIS
LIN {X 50.511,Y 72.808,Z 80.335,A 180.000,B 0.000,C 180.000} C_DIS
LIN {X 50.553,Y 72.875,Z 80.332,A 180.000,B 0.000,C 180.000} C_DIS
LIN {X 50.598,Y 72.940,Z 80.329,A 180.000,B 0.000,C 180.000} C_DIS
LIN {X 50.644,Y 73.004,Z 80.326,A 180.000,B 0.000,C 180.000} C_DIS
LIN {X 50.692,Y 73.066,Z 80.324,A 180.000,B 0.000,C 180.000} C_DIS
LIN {X 50.743,Y 73.126,Z 80.321,A 180.000,B 0.000,C 180.000} C_DIS
LIN {X 50.795,Y 73.185,Z 80.318,A 180.000,B 0.000,C 180.000} C_DIS
LIN {X 50.849,Y 73.243,Z 80.315,A 180.000,B 0.000,C 180.000} C_DIS
LIN {X 50.905,Y 73.298,Z 80.313,A 180.000,B 0.000,C 180.000} C_DIS
LIN {X 50.962,Y 73.352,Z 80.310,A 180.000,B 0.000,C 180.000} C_DIS
LIN {X 51.021,Y 73.404,Z 80.307,A 180.000,B 0.000,C 180.000} C_DIS
LIN {X 51.082,Y 73.454,Z 80.304,A 180.000,B 0.000,C 180.000} C_DIS
LIN {X 51.144,Y 73.502,Z 80.302,A 180.000,B 0.000,C 180.000} C_DIS
LIN {X 51.208,Y 73.549,Z 80.299,A 180.000,B 0.000,C 180.000} C_DIS
LIN {X 51.274,Y 73.593,Z 80.296,A 180.000,B 0.000,C 180.000} C_DIS
LIN {X 51.340,Y 73.635,Z 80.293,A 180.000,B 0.000,C 180.000} C_DIS
LIN {X 51.408,Y 73.675,Z 80.291,A 180.000,B 0.000,C 180.000} C_DIS
LIN {X 51.477,Y 73.712,Z 80.288,A 180.000,B 0.000,C 180.000} C_DIS
LIN {X 51.547,Y 73.748,Z 80.285,A 180.000,B 0.000,C 180.000} C_DIS
LIN {X 51.619,Y 73.781,Z 80.282,A 180.000,B 0.000,C 180.000} C_DIS
LIN {X 51.691,Y 73.812,Z 80.280,A 180.000,B 0.000,C 180.000} C_DIS
LIN {X 51.764,Y 73.841,Z 80.277,A 180.000,B 0.000,C 180.000} C_DIS
LIN {X 51.839,Y 73.868,Z 80.274,A 180.000,B 0.000,C 180.000} C_DIS
LIN {X 51.914,Y 73.892,Z 80.271,A 180.000,B 0.000,C 180.000} C_DIS
LIN {X 51.989,Y 73.913,Z 80.269,A 180.000,B 0.000,C 180.000} C_DIS
LIN {X 52.066,Y 73.933,Z 80.266,A 180.000,B 0.000,C 180.000} C_DIS
LIN {X 52.143,Y 73.950,Z 80.263,A 180.000,B 0.000,C 180.000} C_DIS
LIN {X 52.220,Y 73.964,Z 80.260,A 180.000,B 0.000,C 180.000} C_DIS
LIN {X 52.298,Y 73.976,Z 80.258,A 180.000,B 0.000,C 180.000} C_DIS
LIN {X 52.376,Y 73.986,Z 80.255,A 180.000,B 0.000,C 180.000} C_DIS
LIN {X 52.454,Y 73.993,Z 80.252,A 180.000,B 0.000,C 180.000} C_DIS
LIN {X 52.533,Y 73.998,Z 80.250,A 180.000,B 0.000,C 180.000} C_DIS
LIN {X 52.612,Y 74.000,Z 80.247,A 180.000,B 0.000,C 180.000} C_DIS
LIN {X 52.691,Y 74.000,Z 80.244,A 180.000,B 0.000,C 180.000} C_DIS
LIN {X 52.769,Y 73.997,Z 80.241,A 180.000,B 0.000,C 180.000} C_DIS
LIN {X 52.848,Y 73.991,Z 80.239,A 180.000,B 0.000,C 180.000} C_DIS
LIN {X 52.926,Y 73.984,Z 80.236,A 180.000,B 0.000,C 180.000} C_DIS
LIN {X 53.004,Y 73.973,Z 80.233,A 180.000,B 0.000,C 180.000} C_DIS
LIN {X 53.082,Y 73.961,Z 80.230,A 180.000,B 0.000,C 180.000} C_DIS
LIN {X 53.159,Y 73.946,Z 80.228,A 180.000,B 0.000,C 180.000} C_DIS
LIN {X 53.236,Y 73.928,Z 80.225,A 180.000,B 0.000,C 180.000} C_DIS
LIN {X 53.312,Y 73.908,Z 80.222,A 180.000,B 0.000,C 180.000} C_DIS
LIN {X 53.388,Y 73.886,Z 80.219,A 180.000,B 0.000,C 180.000} C_DIS
LIN {X 53.463,Y 73.861,Z 80.217,A 180.000,B 0.000,C 180.000} C_DIS
LIN {X 53.612,Y 73.811,Z 80.211,A 180.000,B 0.000,C 180.000} C_DIS
LIN {X 53.836,Y 73.735,Z 80.203,A 180.000,B 0.000,C 180.000} C_DIS
LIN {X 53.985,Y 73.685,Z 80.197,A 180.000,B 0.000,C 180.000} C_DIS
LIN {X 54.060,Y 73.660,Z 80.195,A 180.000,B 0.000,C 180.000} C_DIS
LIN {X 54.209,Y 73.610,Z 80.189,A 180.000,B 0.000,C 180.000} C_DIS
LIN {X 54.358,Y 73.559,Z 80.184,A 180.000,B 0.000,C 180.000} C_DIS
LIN {X 54.507,Y 73.509,Z 80.178,A 180.000,B 0.000,C 180.000} C_DIS
LIN {X 54.657,Y 73.459,Z 80.173,A 180.000,B 0.000,C 180.000} C_DIS
LIN {X 54.806,Y 73.408,Z 80.168,A 180.000,B 0.000,C 180.000} C_DIS
LIN {X 54.881,Y 73.383,Z 80.165,A 180.000,B 0.000,C 180.000} C_DIS
LIN {X 54.955,Y 73.358,Z 80.162,A 180.000,B 0.000,C 180.000} C_DIS
LIN {X 55.030,Y 73.333,Z 80.160,A 180.000,B 0.000,C 180.000} C_DIS
LIN {X 55.104,Y 73.308,Z 80.157,A 180.000,B 0.000,C 180.000} C_DIS
LIN {X 55.179,Y 73.282,Z 80.155,A 180.000,B 0.000,C 180.000} C_DIS
LIN {X 55.254,Y 73.257,Z 80.152,A 180.000,B 0.000,C 180.000} C_DIS
LIN {X 55.328,Y 73.232,Z 80.150,A 180.000,B 0.000,C 180.000} C_DIS
LIN {X 55.403,Y 73.207,Z 80.147,A 180.000,B 0.000,C 180.000} C_DIS
LIN {X 55.552,Y 73.156,Z 80.142,A 180.000,B 0.000,C 180.000} C_DIS
LIN {X 55.701,Y 73.106,Z 80.137,A 180.000,B 0.000,C 180.000} C_DIS
LIN {X 55.851,Y 73.056,Z 80.132,A 180.000,B 0.000,C 180.000} C_DIS
LIN {X 56.000,Y 73.005,Z 80.128,A 180.000,B 0.000,C 180.000} C_DIS
LIN {X 56.149,Y 72.955,Z 80.123,A 180.000,B 0.000,C 180.000} C_DIS
LIN {X 56.298,Y 72.905,Z 80.118,A 180.000,B 0.000,C 180.000} C_DIS
LIN {X 56.448,Y 72.854,Z 80.114,A 180.000,B 0.000,C 180.000} C_DIS
LIN {X 56.597,Y 72.804,Z 80.109,A 180.000,B 0.000,C 180.000} C_DIS
LIN {X 56.746,Y 72.754,Z 80.105,A 180.000,B 0.000,C 180.000} C_DIS
LIN {X 56.895,Y 72.703,Z 80.100,A 180.000,B 0.000,C 180.000} C_DIS
LIN {X 57.044,Y 72.653,Z 80.096,A 180.000,B 0.000,C 180.000} C_DIS
LIN {X 57.194,Y 72.603,Z 80.092,A 180.000,B 0.000,C 180.000} C_DIS
LIN {X 57.343,Y 72.552,Z 80.088,A 180.000,B 0.000,C 180.000} C_DIS
LIN {X 57.492,Y 72.502,Z 80.084,A 180.000,B 0.000,C 180.000} C_DIS
LIN {X 57.641,Y 72.452,Z 80.080,A 180.000,B 0.000,C 180.000} C_DIS
LIN {X 57.791,Y 72.401,Z 80.076,A 180.000,B 0.000,C 180.000} C_DIS
LIN {X 57.940,Y 72.351,Z 80.072,A 180.000,B 0.000,C 180.000} C_DIS
LIN {X 58.089,Y 72.301,Z 80.069,A 180.000,B 0.000,C 180.000} C_DIS
LIN {X 58.238,Y 72.250,Z 80.065,A 180.000,B 0.000,C 180.000} C_DIS
LIN {X 58.388,Y 72.200,Z 80.061,A 180.000,B 0.000,C 180.000} C_DIS
LIN {X 58.537,Y 72.150,Z 80.058,A 180.000,B 0.000,C 180.000} C_DIS
LIN {X 58.686,Y 72.099,Z 80.055,A 180.000,B 0.000,C 180.000} C_DIS
LIN {X 58.835,Y 72.049,Z 80.051,A 180.000,B 0.000,C 180.000} C_DIS
LIN {X 58.985,Y 71.999,Z 80.048,A 180.000,B 0.000,C 180.000} C_DIS
LIN {X 59.134,Y 71.948,Z 80.045,A 180.000,B 0.000,C 180.000} C_DIS
LIN {X 59.283,Y 71.898,Z 80.042,A 180.000,B 0.000,C 180.000} C_DIS
LIN {X 59.432,Y 71.848,Z 80.039,A 180.000,B 0.000,C 180.000} C_DIS
LIN {X 59.581,Y 71.797,Z 80.036,A 180.000,B 0.000,C 180.000} C_DIS
LIN {X 59.731,Y 71.747,Z 80.034,A 180.000,B 0.000,C 180.000} C_DIS
LIN {X 59.880,Y 71.696,Z 80.031,A 180.000,B 0.000,C 180.000} C_DIS
LIN {X 60.029,Y 71.646,Z 80.028,A 180.000,B 0.000,C 180.000} C_DIS
LIN {X 60.328,Y 71.545,Z 80.024,A 180.000,B 0.000,C 180.000} C_DIS
LIN {X 60.626,Y 71.445,Z 80.019,A 180.000,B 0.000,C 180.000} C_DIS
LIN {X 60.925,Y 71.344,Z 80.015,A 180.000,B 0.000,C 180.000} C_DIS
LIN {X 61.223,Y 71.243,Z 80.012,A 180.000,B 0.000,C 180.000} C_DIS
LIN {X 61.522,Y 71.143,Z 80.009,A 180.000,B 0.000,C 180.000} C_DIS
LIN {X 61.820,Y 71.042,Z 80.006,A 180.000,B 0.000,C 180.000} C_DIS
LIN {X 62.118,Y 70.941,Z 80.004,A 180.000,B 0.000,C 180.000} C_DIS
LIN {X 62.417,Y 70.841,Z 80.002,A 180.000,B 0.000,C 180.000} C_DIS
LIN {X 62.715,Y 70.740,Z 80.001,A 180.000,B 0.000,C 180.000} C_DIS
LIN {X 63.014,Y 70.639,Z 80.000,A 180.000,B 0.000,C 180.000} C_DIS
LIN {X 63.312,Y 70.539,Z 80.000,A 180.000,B 0.000,C 180.000} C_DIS
LIN {X 63.340,Y 70.529,Z 80.000,A 180.000,B 0.000,C 180.000} C_DIS
; Cutting Move Starts
LIN {X 67.936,Y 68.979,Z 80.000,A 180.000,B 0.000,C 180.000} C_DIS
LIN {X 68.115,Y 68.917,Z 80.000,A 180.000,B 0.000,C 180.000} C_DIS
LIN {X 68.204,Y 68.882,Z 80.000,A 180.000,B 0.000,C 180.000} C_DIS
LIN {X 68.293,Y 68.842,Z 80.000,A 180.000,B 0.000,C 180.000} C_DIS
LIN {X 68.320,Y 68.830,Z 80.000,A 180.000,B 0.000,C 180.000} C_DIS
LIN {X 68.396,Y 68.792,Z 80.000,A 180.000,B 0.000,C 180.000} C_DIS
LIN {X 68.472,Y 68.750,Z 80.000,A 180.000,B 0.000,C 180.000} C_DIS
LIN {X 68.553,Y 68.703,Z 80.000,A 180.000,B 0.000,C 180.000} C_DIS
LIN {X 68.633,Y 68.651,Z 80.000,A 180.000,B 0.000,C 180.000} C_DIS
LIN {X 68.651,Y 68.639,Z 80.000,A 180.000,B 0.000,C 180.000} C_DIS
LIN {X 68.740,Y 68.575,Z 80.000,A 180.000,B 0.000,C 180.000} C_DIS
LIN {X 68.830,Y 68.504,Z 80.000,A 180.000,B 0.000,C 180.000} C_DIS
LIN {X 68.868,Y 68.472,Z 80.000,A 180.000,B 0.000,C 180.000} C_DIS
LIN {X 68.938,Y 68.409,Z 80.000,A 180.000,B 0.000,C 180.000} C_DIS
LIN {X 69.008,Y 68.342,Z 80.000,A 180.000,B 0.000,C 180.000} C_DIS
LIN {X 69.056,Y 68.293,Z 80.000,A 180.000,B 0.000,C 180.000} C_DIS
LIN {X 69.124,Y 68.218,Z 80.000,A 180.000,B 0.000,C 180.000} C_DIS
LIN {X 69.187,Y 68.142,Z 80.000,A 180.000,B 0.000,C 180.000} C_DIS
LIN {X 69.209,Y 68.115,Z 80.000,A 180.000,B 0.000,C 180.000} C_DIS
LIN {X 69.276,Y 68.025,Z 80.000,A 180.000,B 0.000,C 180.000} C_DIS
LIN {X 69.337,Y 67.936,Z 80.000,A 180.000,B 0.000,C 180.000} C_DIS
LIN {X 69.366,Y 67.890,Z 80.000,A 180.000,B 0.000,C 180.000} C_DIS
LIN {X 69.442,Y 67.757,Z 80.000,A 180.000,B 0.000,C 180.000} C_DIS
LIN {X 69.529,Y 67.578,Z 80.000,A 180.000,B 0.000,C 180.000} C_DIS
LIN {X 69.545,Y 67.542,Z 80.000,A 180.000,B 0.000,C 180.000} C_DIS
LIN {X 69.600,Y 67.399,Z 80.000,A 180.000,B 0.000,C 180.000} C_DIS
LIN {X 69.655,Y 67.221,Z 80.000,A 180.000,B 0.000,C 180.000} C_DIS
LIN {X 69.695,Y 67.042,Z 80.000,A 180.000,B 0.000,C 180.000} C_DIS
LIN {X 69.723,Y 66.863,Z 80.000,A 180.000,B 0.000,C 180.000} C_DIS
LIN {X 69.724,Y 66.856,Z 80.000,A 180.000,B 0.000,C 180.000} C_DIS
LIN {X 69.737,Y 66.684,Z 80.000,A 180.000,B 0.000,C 180.000} C_DIS
LIN {X 69.738,Y 66.506,Z 80.000,A 180.000,B 0.000,C 180.000} C_DIS
LIN {X 69.727,Y 66.327,Z 80.000,A 180.000,B 0.000,C 180.000} C_DIS
LIN {X 69.724,Y 66.295,Z 80.000,A 180.000,B 0.000,C 180.000} C_DIS
LIN {X 69.703,Y 66.148,Z 80.000,A 180.000,B 0.000,C 180.000} C_DIS
LIN {X 69.665,Y 65.969,Z 80.000,A 180.000,B 0.000,C 180.000} C_DIS
LIN {X 69.613,Y 65.791,Z 80.000,A 180.000,B 0.000,C 180.000} C_DIS
LIN {X 69.553,Y 65.612,Z 80.000,A 180.000,B 0.000,C 180.000} C_DIS
LIN {X 63.220,Y 46.841,Z 80.000,A 180.000,B 0.000,C 180.000} C_DIS
LIN {X 63.154,Y 46.662,Z 80.000,A 180.000,B 0.000,C 180.000} C_DIS
LIN {X 63.109,Y 46.562,Z 80.000,A 180.000,B 0.000,C 180.000} C_DIS
LIN {X 63.071,Y 46.483,Z 80.000,A 180.000,B 0.000,C 180.000} C_DIS
LIN {X 62.969,Y 46.305,Z 80.000,A 180.000,B 0.000,C 180.000} C_DIS
LIN {X 62.930,Y 46.244,Z 80.000,A 180.000,B 0.000,C 180.000} C_DIS
LIN {X 62.847,Y 46.126,Z 80.000,A 180.000,B 0.000,C 180.000} C_DIS
LIN {X 62.751,Y 46.006,Z 80.000,A 180.000,B 0.000,C 180.000} C_DIS
LIN {X 62.700,Y 45.947,Z 80.000,A 180.000,B 0.000,C 180.000} C_DIS
LIN {X 62.573,Y 45.816,Z 80.000,A 180.000,B 0.000,C 180.000} C_DIS
LIN {X 62.521,Y 45.768,Z 80.000,A 180.000,B 0.000,C 180.000} C_DIS
LIN {X 62.394,Y 45.661,Z 80.000,A 180.000,B 0.000,C 180.000} C_DIS
LIN {X 62.298,Y 45.590,Z 80.000,A 180.000,B 0.000,C 180.000} C_DIS
LIN {X 62.215,Y 45.533,Z 80.000,A 180.000,B 0.000,C 180.000} C_DIS
LIN {X 62.036,Y 45.426,Z 80.000,A 180.000,B 0.000,C 180.000} C_DIS
LIN {X 62.008,Y 45.411,Z 80.000,A 180.000,B 0.000,C 180.000} C_DIS
LIN {X 61.858,Y 45.338,Z 80.000,A 180.000,B 0.000,C 180.000} C_DIS
LIN {X 61.679,Y 45.267,Z 80.000,A 180.000,B 0.000,C 180.000} C_DIS
LIN {X 61.571,Y 45.232,Z 80.000,A 180.000,B 0.000,C 180.000} C_DIS
LIN {X 61.500,Y 45.212,Z 80.000,A 180.000,B 0.000,C 180.000} C_DIS
LIN {X 61.321,Y 45.170,Z 80.000,A 180.000,B 0.000,C 180.000} C_DIS
LIN {X 61.232,Y 45.155,Z 80.000,A 180.000,B 0.000,C 180.000} C_DIS
LIN {X 61.143,Y 45.142,Z 80.000,A 180.000,B 0.000,C 180.000} C_DIS
LIN {X 61.053,Y 45.133,Z 80.000,A 180.000,B 0.000,C 180.000} C_DIS
LIN {X 60.964,Y 45.127,Z 80.000,A 180.000,B 0.000,C 180.000} C_DIS
LIN {X 60.874,Y 45.125,Z 80.000,A 180.000,B 0.000,C 180.000} C_DIS
LIN {X 60.785,Y 45.125,Z 80.000,A 180.000,B 0.000,C 180.000} C_DIS
LIN {X 60.696,Y 45.129,Z 80.000,A 180.000,B 0.000,C 180.000} C_DIS
LIN {X 60.606,Y 45.136,Z 80.000,A 180.000,B 0.000,C 180.000} C_DIS
LIN {X 60.517,Y 45.146,Z 80.000,A 180.000,B 0.000,C 180.000} C_DIS
LIN {X 60.427,Y 45.160,Z 80.000,A 180.000,B 0.000,C 180.000} C_DIS
LIN {X 60.338,Y 45.177,Z 80.000,A 180.000,B 0.000,C 180.000} C_DIS
LIN {X 60.249,Y 45.197,Z 80.000,A 180.000,B 0.000,C 180.000} C_DIS
LIN {X 60.185,Y 45.214,Z 80.000,A 180.000,B 0.000,C 180.000} C_DIS
LIN {X 60.122,Y 45.232,Z 80.000,A 180.000,B 0.000,C 180.000} C_DIS
LIN {X 60.070,Y 45.248,Z 80.000,A 180.000,B 0.000,C 180.000} C_DIS
LIN {X 59.891,Y 45.308,Z 80.000,A 180.000,B 0.000,C 180.000} C_DIS
LIN {X 45.590,Y 50.133,Z 80.000,A 180.000,B 0.000,C 180.000} C_DIS
LIN {X 45.411,Y 50.194,Z 80.000,A 180.000,B 0.000,C 180.000} C_DIS
LIN {X 45.296,Y 50.238,Z 80.000,A 180.000,B 0.000,C 180.000} C_DIS
LIN {X 45.232,Y 50.265,Z 80.000,A 180.000,B 0.000,C 180.000} C_DIS
LIN {X 45.053,Y 50.353,Z 80.000,A 180.000,B 0.000,C 180.000} C_DIS
LIN {X 44.944,Y 50.416,Z 80.000,A 180.000,B 0.000,C 180.000} C_DIS
LIN {X 44.874,Y 50.461,Z 80.000,A 180.000,B 0.000,C 180.000} C_DIS
LIN {X 44.785,Y 50.522,Z 80.000,A 180.000,B 0.000,C 180.000} C_DIS
LIN {X 44.696,Y 50.590,Z 80.000,A 180.000,B 0.000,C 180.000} C_DIS
LIN {X 44.689,Y 50.595,Z 80.000,A 180.000,B 0.000,C 180.000} C_DIS
LIN {X 44.603,Y 50.667,Z 80.000,A 180.000,B 0.000,C 180.000} C_DIS
LIN {X 44.517,Y 50.746,Z 80.000,A 180.000,B 0.000,C 180.000} C_DIS
LIN {X 44.488,Y 50.774,Z 80.000,A 180.000,B 0.000,C 180.000} C_DIS
LIN {X 44.410,Y 50.855,Z 80.000,A 180.000,B 0.000,C 180.000} C_DIS
LIN {X 44.338,Y 50.936,Z 80.000,A 180.000,B 0.000,C 180.000} C_DIS
LIN {X 44.325,Y 50.953,Z 80.000,A 180.000,B 0.000,C 180.000} C_DIS
LIN {X 44.254,Y 51.042,Z 80.000,A 180.000,B 0.000,C 180.000} C_DIS
LIN {X 44.189,Y 51.131,Z 80.000,A 180.000,B 0.000,C 180.000} C_DIS
LIN {X 44.159,Y 51.176,Z 80.000,A 180.000,B 0.000,C 180.000} C_DIS
LIN {X 44.077,Y 51.310,Z 80.000,A 180.000,B 0.000,C 180.000} C_DIS
LIN {X 43.984,Y 51.489,Z 80.000,A 180.000,B 0.000,C 180.000} C_DIS
LIN {X 43.981,Y 51.497,Z 80.000,A 180.000,B 0.000,C 180.000} C_DIS
LIN {X 43.909,Y 51.668,Z 80.000,A 180.000,B 0.000,C 180.000} C_DIS
LIN {X 43.849,Y 51.847,Z 80.000,A 180.000,B 0.000,C 180.000} C_DIS
LIN {X 43.804,Y 52.025,Z 80.000,A 180.000,B 0.000,C 180.000} C_DIS
LIN {X 43.802,Y 52.035,Z 80.000,A 180.000,B 0.000,C 180.000} C_DIS
LIN {X 43.772,Y 52.204,Z 80.000,A 180.000,B 0.000,C 180.000} C_DIS
LIN {X 43.754,Y 52.383,Z 80.000,A 180.000,B 0.000,C 180.000} C_DIS
LIN {X 43.748,Y 52.562,Z 80.000,A 180.000,B 0.000,C 180.000} C_DIS
LIN {X 43.756,Y 52.740,Z 80.000,A 180.000,B 0.000,C 180.000} C_DIS
LIN {X 43.776,Y 52.919,Z 80.000,A 180.000,B 0.000,C 180.000} C_DIS
LIN {X 43.802,Y 53.064,Z 80.000,A 180.000,B 0.000,C 180.000} C_DIS
LIN {X 43.809,Y 53.098,Z 80.000,A 180.000,B 0.000,C 180.000} C_DIS
LIN {X 43.856,Y 53.277,Z 80.000,A 180.000,B 0.000,C 180.000} C_DIS
LIN {X 43.916,Y 53.455,Z 80.000,A 180.000,B 0.000,C 180.000} C_DIS
LIN {X 50.248,Y 72.226,Z 80.000,A 180.000,B 0.000,C 180.000} C_DIS
LIN {X 50.311,Y 72.405,Z 80.000,A 180.000,B 0.000,C 180.000} C_DIS
LIN {X 50.388,Y 72.584,Z 80.000,A 180.000,B 0.000,C 180.000} C_DIS
LIN {X 50.416,Y 72.640,Z 80.000,A 180.000,B 0.000,C 180.000} C_DIS
LIN {X 50.484,Y 72.763,Z 80.000,A 180.000,B 0.000,C 180.000} C_DIS
LIN {X 50.595,Y 72.936,Z 80.000,A 180.000,B 0.000,C 180.000} C_DIS
LIN {X 50.599,Y 72.941,Z 80.000,A 180.000,B 0.000,C 180.000} C_DIS
LIN {X 50.665,Y 73.031,Z 80.000,A 180.000,B 0.000,C 180.000} C_DIS
LIN {X 50.737,Y 73.120,Z 80.000,A 180.000,B 0.000,C 180.000} C_DIS
LIN {X 50.774,Y 73.162,Z 80.000,A 180.000,B 0.000,C 180.000} C_DIS
LIN {X 50.905,Y 73.299,Z 80.000,A 180.000,B 0.000,C 180.000} C_DIS
LIN {X 50.953,Y 73.343,Z 80.000,A 180.000,B 0.000,C 180.000} C_DIS
LIN {X 51.112,Y 73.478,Z 80.000,A 180.000,B 0.000,C 180.000} C_DIS
LIN {X 51.131,Y 73.493,Z 80.000,A 180.000,B 0.000,C 180.000} C_DIS
LIN {X 51.310,Y 73.616,Z 80.000,A 180.000,B 0.000,C 180.000} C_DIS
LIN {X 51.376,Y 73.656,Z 80.000,A 180.000,B 0.000,C 180.000} C_DIS
LIN {X 51.489,Y 73.719,Z 80.000,A 180.000,B 0.000,C 180.000} C_DIS
LIN {X 51.668,Y 73.803,Z 80.000,A 180.000,B 0.000,C 180.000} C_DIS
LIN {X 51.749,Y 73.835,Z 80.000,A 180.000,B 0.000,C 180.000} C_DIS
LIN {X 51.847,Y 73.870,Z 80.000,A 180.000,B 0.000,C 180.000} C_DIS
LIN {X 52.025,Y 73.923,Z 80.000,A 180.000,B 0.000,C 180.000} C_DIS
LIN {X 52.204,Y 73.961,Z 80.000,A 180.000,B 0.000,C 180.000} C_DIS
LIN {X 52.383,Y 73.987,Z 80.000,A 180.000,B 0.000,C 180.000} C_DIS
LIN {X 52.562,Y 73.999,Z 80.000,A 180.000,B 0.000,C 180.000} C_DIS
LIN {X 52.740,Y 73.998,Z 80.000,A 180.000,B 0.000,C 180.000} C_DIS
LIN {X 52.919,Y 73.985,Z 80.000,A 180.000,B 0.000,C 180.000} C_DIS
LIN {X 53.098,Y 73.958,Z 80.000,A 180.000,B 0.000,C 180.000} C_DIS
LIN {X 53.277,Y 73.918,Z 80.000,A 180.000,B 0.000,C 180.000} C_DIS
LIN {X 53.455,Y 73.864,Z 80.000,A 180.000,B 0.000,C 180.000} C_DIS
LIN {X 63.340,Y 70.529,Z 80.000,A 180.000,B 0.000,C 180.000} C_DIS
; Link Move Starts
LIN {X 63.639,Y 70.428,Z 80.000,A 180.000,B 0.000,C 180.000} C_DIS
LIN {X 63.937,Y 70.328,Z 79.999,A 180.000,B 0.000,C 180.000} C_DIS
LIN {X 64.236,Y 70.227,Z 79.998,A 180.000,B 0.000,C 180.000} C_DIS
LIN {X 64.534,Y 70.126,Z 79.996,A 180.000,B 0.000,C 180.000} C_DIS
LIN {X 64.833,Y 70.026,Z 79.994,A 180.000,B 0.000,C 180.000} C_DIS
LIN {X 65.131,Y 69.925,Z 79.991,A 180.000,B 0.000,C 180.000} C_DIS
LIN {X 65.429,Y 69.824,Z 79.988,A 180.000,B 0.000,C 180.000} C_DIS
LIN {X 65.728,Y 69.724,Z 79.985,A 180.000,B 0.000,C 180.000} C_DIS
LIN {X 66.026,Y 69.623,Z 79.981,A 180.000,B 0.000,C 180.000} C_DIS
LIN {X 66.325,Y 69.522,Z 79.977,A 180.000,B 0.000,C 180.000} C_DIS
LIN {X 66.623,Y 69.422,Z 79.972,A 180.000,B 0.000,C 180.000} C_DIS
LIN {X 66.773,Y 69.371,Z 79.969,A 180.000,B 0.000,C 180.000} C_DIS
LIN {X 66.922,Y 69.321,Z 79.967,A 180.000,B 0.000,C 180.000} C_DIS
LIN {X 67.071,Y 69.271,Z 79.964,A 180.000,B 0.000,C 180.000} C_DIS
LIN {X 67.220,Y 69.220,Z 79.961,A 180.000,B 0.000,C 180.000} C_DIS
LIN {X 67.370,Y 69.170,Z 79.959,A 180.000,B 0.000,C 180.000} C_DIS
LIN {X 67.519,Y 69.120,Z 79.956,A 180.000,B 0.000,C 180.000} C_DIS
LIN {X 67.668,Y 69.069,Z 79.952,A 180.000,B 0.000,C 180.000} C_DIS
LIN {X 67.817,Y 69.019,Z 79.949,A 180.000,B 0.000,C 180.000} C_DIS
LIN {X 67.967,Y 68.968,Z 79.946,A 180.000,B 0.000,C 180.000} C_DIS
LIN {X 68.116,Y 68.918,Z 79.943,A 180.000,B 0.000,C 180.000} C_DIS
LIN {X 68.190,Y 68.892,Z 79.941,A 180.000,B 0.000,C 180.000} C_DIS
LIN {X 68.264,Y 68.863,Z 79.939,A 180.000,B 0.000,C 180.000} C_DIS
LIN {X 68.336,Y 68.832,Z 79.937,A 180.000,B 0.000,C 180.000} C_DIS
LIN {X 68.408,Y 68.799,Z 79.936,A 180.000,B 0.000,C 180.000} C_DIS
LIN {X 68.480,Y 68.764,Z 79.934,A 180.000,B 0.000,C 180.000} C_DIS
LIN {X 68.550,Y 68.726,Z 79.932,A 180.000,B 0.000,C 180.000} C_DIS
LIN {X 68.620,Y 68.686,Z 79.930,A 180.000,B 0.000,C 180.000} C_DIS
LIN {X 68.688,Y 68.644,Z 79.928,A 180.000,B 0.000,C 180.000} C_DIS
LIN {X 68.757,Y 68.599,Z 79.926,A 180.000,B 0.000,C 180.000} C_DIS
LIN {X 68.825,Y 68.551,Z 79.924,A 180.000,B 0.000,C 180.000} C_DIS
LIN {X 68.891,Y 68.502,Z 79.922,A 180.000,B 0.000,C 180.000} C_DIS
LIN {X 68.955,Y 68.450,Z 79.920,A 180.000,B 0.000,C 180.000} C_DIS
LIN {X 69.084,Y 68.337,Z 79.916,A 180.000,B 0.000,C 180.000} C_DIS
LIN {X 69.205,Y 68.216,Z 79.911,A 180.000,B 0.000,C 180.000} C_DIS
LIN {X 69.304,Y 68.105,Z 79.907,A 180.000,B 0.000,C 180.000} C_DIS
LIN {X 69.397,Y 67.988,Z 79.903,A 180.000,B 0.000,C 180.000} C_DIS
LIN {X 69.477,Y 67.875,Z 79.900,A 180.000,B 0.000,C 180.000} C_DIS
LIN {X 69.550,Y 67.758,Z 79.896,A 180.000,B 0.000,C 180.000} C_DIS
LIN {X 69.614,Y 67.645,Z 79.892,A 180.000,B 0.000,C 180.000} C_DIS
LIN {X 69.673,Y 67.530,Z 79.888,A 180.000,B 0.000,C 180.000} C_DIS
LIN {X 69.720,Y 67.424,Z 79.885,A 180.000,B 0.000,C 180.000} C_DIS
LIN {X 69.763,Y 67.316,Z 79.881,A 180.000,B 0.000,C 180.000} C_DIS
LIN {X 69.800,Y 67.208,Z 79.878,A 180.000,B 0.000,C 180.000} C_DIS
LIN {X 69.833,Y 67.098,Z 79.874,A 180.000,B 0.000,C 180.000} C_DIS
LIN {X 69.861,Y 66.987,Z 79.871,A 180.000,B 0.000,C 180.000} C_DIS
LIN {X 69.884,Y 66.876,Z 79.867,A 180.000,B 0.000,C 180.000} C_DIS
LIN {X 69.898,Y 66.790,Z 79.864,A 180.000,B 0.000,C 180.000} C_DIS
LIN {X 69.910,Y 66.704,Z 79.861,A 180.000,B 0.000,C 180.000} C_DIS
LIN {X 69.921,Y 66.590,Z 79.857,A 180.000,B 0.000,C 180.000} C_DIS
LIN {X 69.926,Y 66.476,Z 79.854,A 180.000,B 0.000,C 180.000} C_DIS
LIN {X 69.927,Y 66.382,Z 79.851,A 180.000,B 0.000,C 180.000} C_DIS
LIN {X 69.925,Y 66.289,Z 79.847,A 180.000,B 0.000,C 180.000} C_DIS
LIN {X 69.920,Y 66.206,Z 79.844,A 180.000,B 0.000,C 180.000} C_DIS
LIN {X 69.913,Y 66.124,Z 79.842,A 180.000,B 0.000,C 180.000} C_DIS
LIN {X 69.901,Y 66.034,Z 79.838,A 180.000,B 0.000,C 180.000} C_DIS
LIN {X 69.887,Y 65.945,Z 79.835,A 180.000,B 0.000,C 180.000} C_DIS
LIN {X 69.866,Y 65.843,Z 79.832,A 180.000,B 0.000,C 180.000} C_DIS
LIN {X 69.841,Y 65.741,Z 79.828,A 180.000,B 0.000,C 180.000} C_DIS
LIN {X 69.807,Y 65.620,Z 79.824,A 180.000,B 0.000,C 180.000} C_DIS
LIN {X 69.772,Y 65.498,Z 79.819,A 180.000,B 0.000,C 180.000} C_DIS
LIN {X 69.750,Y 65.422,Z 79.816,A 180.000,B 0.000,C 180.000} C_DIS
LIN {X 69.729,Y 65.347,Z 79.814,A 180.000,B 0.000,C 180.000} C_DIS
LIN {X 69.707,Y 65.271,Z 79.811,A 180.000,B 0.000,C 180.000} C_DIS
LIN {X 69.685,Y 65.195,Z 79.808,A 180.000,B 0.000,C 180.000} C_DIS
LIN {X 69.664,Y 65.119,Z 79.806,A 180.000,B 0.000,C 180.000} C_DIS
LIN {X 69.642,Y 65.043,Z 79.803,A 180.000,B 0.000,C 180.000} C_DIS
LIN {X 69.620,Y 64.968,Z 79.800,A 180.000,B 0.000,C 180.000} C_DIS
LIN {X 69.599,Y 64.892,Z 79.797,A 180.000,B 0.000,C 180.000} C_DIS
LIN {X 69.577,Y 64.816,Z 79.795,A 180.000,B 0.000,C 180.000} C_DIS
LIN {X 69.555,Y 64.740,Z 79.792,A 180.000,B 0.000,C 180.000} C_DIS
LIN {X 69.534,Y 64.664,Z 79.789,A 180.000,B 0.000,C 180.000} C_DIS
LIN {X 69.512,Y 64.589,Z 79.786,A 180.000,B 0.000,C 180.000} C_DIS
LIN {X 69.491,Y 64.513,Z 79.784,A 180.000,B 0.000,C 180.000} C_DIS
LIN {X 69.469,Y 64.437,Z 79.781,A 180.000,B 0.000,C 180.000} C_DIS
LIN {X 69.447,Y 64.361,Z 79.778,A 180.000,B 0.000,C 180.000} C_DIS
LIN {X 69.426,Y 64.285,Z 79.775,A 180.000,B 0.000,C 180.000} C_DIS
LIN {X 69.404,Y 64.209,Z 79.773,A 180.000,B 0.000,C 180.000} C_DIS
LIN {X 69.382,Y 64.134,Z 79.770,A 180.000,B 0.000,C 180.000} C_DIS
LIN {X 69.361,Y 64.058,Z 79.767,A 180.000,B 0.000,C 180.000} C_DIS
LIN {X 69.339,Y 63.982,Z 79.764,A 180.000,B 0.000,C 180.000} C_DIS
LIN {X 69.317,Y 63.906,Z 79.761,A 180.000,B 0.000,C 180.000} C_DIS
LIN {X 69.296,Y 63.830,Z 79.759,A 180.000,B 0.000,C 180.000} C_DIS
LIN {X 69.274,Y 63.755,Z 79.756,A 180.000,B 0.000,C 180.000} C_DIS
LIN {X 69.252,Y 63.679,Z 79.753,A 180.000,B 0.000,C 180.000} C_DIS
LIN {X 69.231,Y 63.603,Z 79.750,A 180.000,B 0.000,C 180.000} C_DIS
LIN {X 69.209,Y 63.527,Z 79.748,A 180.000,B 0.000,C 180.000} C_DIS
LIN {X 69.144,Y 63.300,Z 79.739,A 180.000,B 0.000,C 180.000} C_DIS
LIN {X 69.101,Y 63.148,Z 79.734,A 180.000,B 0.000,C 180.000} C_DIS
LIN {X 69.079,Y 63.072,Z 79.731,A 180.000,B 0.000,C 180.000} C_DIS
LIN {X 69.036,Y 62.921,Z 79.726,A 180.000,B 0.000,C 180.000} C_DIS
LIN {X 68.971,Y 62.693,Z 79.717,A 180.000,B 0.000,C 180.000} C_DIS
LIN {X 68.928,Y 62.542,Z 79.712,A 180.000,B 0.000,C 180.000} C_DIS
LIN {X 68.906,Y 62.466,Z 79.709,A 180.000,B 0.000,C 180.000} C_DIS
LIN {X 68.863,Y 62.314,Z 79.704,A 180.000,B 0.000,C 180.000} C_DIS
LIN {X 68.841,Y 62.238,Z 79.701,A 180.000,B 0.000,C 180.000} C_DIS
LIN {X 68.819,Y 62.163,Z 79.698,A 180.000,B 0.000,C 180.000} C_DIS
LIN {X 68.776,Y 62.011,Z 79.693,A 180.000,B 0.000,C 180.000} C_DIS
LIN {X 68.710,Y 61.784,Z 79.684,A 180.000,B 0.000,C 180.000} C_DIS
LIN {X 68.667,Y 61.632,Z 79.679,A 180.000,B 0.000,C 180.000} C_DIS
LIN {X 68.645,Y 61.557,Z 79.676,A 180.000,B 0.000,C 180.000} C_DIS
LIN {X 68.601,Y 61.405,Z 79.671,A 180.000,B 0.000,C 180.000} C_DIS
LIN {X 68.536,Y 61.178,Z 79.662,A 180.000,B 0.000,C 180.000} C_DIS
LIN {X 68.492,Y 61.026,Z 79.657,A 180.000,B 0.000,C 180.000} C_DIS
LIN {X 68.471,Y 60.951,Z 79.654,A 180.000,B 0.000,C 180.000} C_DIS
LIN {X 68.427,Y 60.799,Z 79.649,A 180.000,B 0.000,C 180.000} C_DIS
LIN {X 68.296,Y 60.345,Z 79.632,A 180.000,B 0.000,C 180.000} C_DIS
LIN {X 68.253,Y 60.193,Z 79.627,A 180.000,B 0.000,C 180.000} C_DIS
LIN {X 68.122,Y 59.738,Z 79.610,A 180.000,B 0.000,C 180.000} C_DIS
LIN {X 68.057,Y 59.511,Z 79.602,A 180.000,B 0.000,C 180.000} C_DIS
LIN {X 68.013,Y 59.360,Z 79.596,A 180.000,B 0.000,C 180.000} C_DIS
LIN {X 67.882,Y 58.905,Z 79.580,A 180.000,B 0.000,C 180.000} C_DIS
LIN {X 67.839,Y 58.754,Z 79.574,A 180.000,B 0.000,C 180.000} C_DIS
LIN {X 67.708,Y 58.299,Z 79.558,A 180.000,B 0.000,C 180.000} C_DIS
LIN {X 67.642,Y 58.072,Z 79.549,A 180.000,B 0.000,C 180.000} C_DIS
LIN {X 67.294,Y 56.860,Z 79.505,A 180.000,B 0.000,C 180.000} C_DIS
LIN {X 66.945,Y 55.648,Z 79.461,A 180.000,B 0.000,C 180.000} C_DIS
LIN {X 66.531,Y 54.208,Z 79.409,A 180.000,B 0.000,C 180.000} C_DIS
LIN {X 66.400,Y 53.754,Z 79.393,A 180.000,B 0.000,C 180.000} C_DIS
LIN {X 66.378,Y 53.678,Z 79.390,A 180.000,B 0.000,C 180.000} C_DIS
LIN {X 66.335,Y 53.526,Z 79.384,A 180.000,B 0.000,C 180.000} C_DIS
LIN {X 66.204,Y 53.072,Z 79.368,A 180.000,B 0.000,C 180.000} C_DIS
LIN {X 66.160,Y 52.920,Z 79.362,A 180.000,B 0.000,C 180.000} C_DIS
LIN {X 66.030,Y 52.466,Z 79.346,A 180.000,B 0.000,C 180.000} C_DIS
LIN {X 65.986,Y 52.314,Z 79.340,A 180.000,B 0.000,C 180.000} C_DIS
LIN {X 65.921,Y 52.087,Z 79.332,A 180.000,B 0.000,C 180.000} C_DIS
LIN {X 65.877,Y 51.935,Z 79.326,A 180.000,B 0.000,C 180.000} C_DIS
LIN {X 65.855,Y 51.860,Z 79.324,A 180.000,B 0.000,C 180.000} C_DIS
LIN {X 65.812,Y 51.708,Z 79.318,A 180.000,B 0.000,C 180.000} C_DIS
LIN {X 65.746,Y 51.481,Z 79.310,A 180.000,B 0.000,C 180.000} C_DIS
LIN {X 65.703,Y 51.329,Z 79.304,A 180.000,B 0.000,C 180.000} C_DIS
LIN {X 65.681,Y 51.254,Z 79.302,A 180.000,B 0.000,C 180.000} C_DIS
LIN {X 65.637,Y 51.102,Z 79.296,A 180.000,B 0.000,C 180.000} C_DIS
LIN {X 65.572,Y 50.875,Z 79.288,A 180.000,B 0.000,C 180.000} C_DIS
LIN {X 65.528,Y 50.723,Z 79.282,A 180.000,B 0.000,C 180.000} C_DIS
LIN {X 65.506,Y 50.648,Z 79.280,A 180.000,B 0.000,C 180.000} C_DIS
LIN {X 65.463,Y 50.496,Z 79.274,A 180.000,B 0.000,C 180.000} C_DIS
LIN {X 65.441,Y 50.420,Z 79.271,A 180.000,B 0.000,C 180.000} C_DIS
LIN {X 65.419,Y 50.345,Z 79.269,A 180.000,B 0.000,C 180.000} C_DIS
LIN {X 65.375,Y 50.193,Z 79.263,A 180.000,B 0.000,C 180.000} C_DIS
LIN {X 65.310,Y 49.966,Z 79.255,A 180.000,B 0.000,C 180.000} C_DIS
LIN {X 65.266,Y 49.815,Z 79.249,A 180.000,B 0.000,C 180.000} C_DIS
LIN {X 65.244,Y 49.739,Z 79.247,A 180.000,B 0.000,C 180.000} C_DIS
LIN {X 65.222,Y 49.663,Z 79.244,A 180.000,B 0.000,C 180.000} C_DIS
LIN {X 65.200,Y 49.587,Z 79.241,A 180.000,B 0.000,C 180.000} C_DIS
LIN {X 65.178,Y 49.512,Z 79.238,A 180.000,B 0.000,C 180.000} C_DIS
LIN {X 65.156,Y 49.436,Z 79.236,A 180.000,B 0.000,C 180.000} C_DIS
LIN {X 65.134,Y 49.360,Z 79.233,A 180.000,B 0.000,C 180.000} C_DIS
LIN {X 65.112,Y 49.285,Z 79.230,A 180.000,B 0.000,C 180.000} C_DIS
LIN {X 65.090,Y 49.209,Z 79.227,A 180.000,B 0.000,C 180.000} C_DIS
LIN {X 65.069,Y 49.133,Z 79.225,A 180.000,B 0.000,C 180.000} C_DIS
LIN {X 65.047,Y 49.057,Z 79.222,A 180.000,B 0.000,C 180.000} C_DIS
LIN {X 65.025,Y 48.982,Z 79.219,A 180.000,B 0.000,C 180.000} C_DIS
LIN {X 65.003,Y 48.906,Z 79.216,A 180.000,B 0.000,C 180.000} C_DIS
LIN {X 64.981,Y 48.830,Z 79.214,A 180.000,B 0.000,C 180.000} C_DIS
LIN {X 64.959,Y 48.755,Z 79.211,A 180.000,B 0.000,C 180.000} C_DIS
LIN {X 64.937,Y 48.679,Z 79.208,A 180.000,B 0.000,C 180.000} C_DIS
LIN {X 64.915,Y 48.603,Z 79.205,A 180.000,B 0.000,C 180.000} C_DIS
LIN {X 64.893,Y 48.527,Z 79.203,A 180.000,B 0.000,C 180.000} C_DIS
LIN {X 64.871,Y 48.452,Z 79.200,A 180.000,B 0.000,C 180.000} C_DIS
LIN {X 64.849,Y 48.376,Z 79.197,A 180.000,B 0.000,C 180.000} C_DIS
LIN {X 64.827,Y 48.300,Z 79.194,A 180.000,B 0.000,C 180.000} C_DIS
LIN {X 64.806,Y 48.225,Z 79.192,A 180.000,B 0.000,C 180.000} C_DIS
LIN {X 64.784,Y 48.149,Z 79.189,A 180.000,B 0.000,C 180.000} C_DIS
LIN {X 64.762,Y 48.073,Z 79.186,A 180.000,B 0.000,C 180.000} C_DIS
LIN {X 64.740,Y 47.997,Z 79.183,A 180.000,B 0.000,C 180.000} C_DIS
LIN {X 64.718,Y 47.922,Z 79.181,A 180.000,B 0.000,C 180.000} C_DIS
LIN {X 64.696,Y 47.846,Z 79.178,A 180.000,B 0.000,C 180.000} C_DIS
LIN {X 64.674,Y 47.770,Z 79.175,A 180.000,B 0.000,C 180.000} C_DIS
LIN {X 64.652,Y 47.695,Z 79.173,A 180.000,B 0.000,C 180.000} C_DIS
LIN {X 64.630,Y 47.619,Z 79.170,A 180.000,B 0.000,C 180.000} C_DIS
LIN {X 64.608,Y 47.543,Z 79.167,A 180.000,B 0.000,C 180.000} C_DIS
LIN {X 64.586,Y 47.468,Z 79.165,A 180.000,B 0.000,C 180.000} C_DIS
LIN {X 64.563,Y 47.392,Z 79.162,A 180.000,B 0.000,C 180.000} C_DIS
LIN {X 64.541,Y 47.316,Z 79.160,A 180.000,B 0.000,C 180.000} C_DIS
LIN {X 64.519,Y 47.241,Z 79.157,A 180.000,B 0.000,C 180.000} C_DIS
LIN {X 64.497,Y 47.165,Z 79.154,A 180.000,B 0.000,C 180.000} C_DIS
LIN {X 64.475,Y 47.089,Z 79.152,A 180.000,B 0.000,C 180.000} C_DIS
LIN {X 64.453,Y 47.014,Z 79.149,A 180.000,B 0.000,C 180.000} C_DIS
LIN {X 64.408,Y 46.863,Z 79.144,A 180.000,B 0.000,C 180.000} C_DIS
LIN {X 64.364,Y 46.711,Z 79.139,A 180.000,B 0.000,C 180.000} C_DIS
LIN {X 64.319,Y 46.561,Z 79.135,A 180.000,B 0.000,C 180.000} C_DIS
LIN {X 64.275,Y 46.411,Z 79.130,A 180.000,B 0.000,C 180.000} C_DIS
LIN {X 64.226,Y 46.274,Z 79.126,A 180.000,B 0.000,C 180.000} C_DIS
LIN {X 64.169,Y 46.139,Z 79.122,A 180.000,B 0.000,C 180.000} C_DIS
LIN {X 64.102,Y 46.005,Z 79.118,A 180.000,B 0.000,C 180.000} C_DIS
LIN {X 64.028,Y 45.875,Z 79.114,A 180.000,B 0.000,C 180.000} C_DIS
LIN {X 63.946,Y 45.752,Z 79.110,A 180.000,B 0.000,C 180.000} C_DIS
LIN {X 63.858,Y 45.633,Z 79.106,A 180.000,B 0.000,C 180.000} C_DIS
LIN {X 63.759,Y 45.517,Z 79.102,A 180.000,B 0.000,C 180.000} C_DIS
LIN {X 63.653,Y 45.408,Z 79.098,A 180.000,B 0.000,C 180.000} C_DIS
LIN {X 63.541,Y 45.306,Z 79.094,A 180.000,B 0.000,C 180.000} C_DIS
LIN {X 63.423,Y 45.211,Z 79.090,A 180.000,B 0.000,C 180.000} C_DIS
LIN {X 63.299,Y 45.123,Z 79.086,A 180.000,B 0.000,C 180.000} C_DIS
LIN {X 63.169,Y 45.044,Z 79.083,A 180.000,B 0.000,C 180.000} C_DIS
LIN {X 63.034,Y 44.972,Z 79.079,A 180.000,B 0.000,C 180.000} C_DIS
LIN {X 62.894,Y 44.910,Z 79.076,A 180.000,B 0.000,C 180.000} C_DIS
LIN {X 62.749,Y 44.855,Z 79.072,A 180.000,B 0.000,C 180.000} C_DIS
LIN {X 62.600,Y 44.811,Z 79.068,A 180.000,B 0.000,C 180.000} C_DIS
LIN {X 62.449,Y 44.776,Z 79.065,A 180.000,B 0.000,C 180.000} C_DIS
LIN {X 62.296,Y 44.751,Z 79.062,A 180.000,B 0.000,C 180.000} C_DIS
LIN {X 62.141,Y 44.736,Z 79.058,A 180.000,B 0.000,C 180.000} C_DIS
LIN {X 61.985,Y 44.731,Z 79.055,A 180.000,B 0.000,C 180.000} C_DIS
LIN {X 61.907,Y 44.733,Z 79.053,A 180.000,B 0.000,C 180.000} C_DIS
LIN {X 61.829,Y 44.737,Z 79.052,A 180.000,B 0.000,C 180.000} C_DIS
LIN {X 61.751,Y 44.744,Z 79.050,A 180.000,B 0.000,C 180.000} C_DIS
LIN {X 61.673,Y 44.753,Z 79.049,A 180.000,B 0.000,C 180.000} C_DIS
LIN {X 61.595,Y 44.765,Z 79.047,A 180.000,B 0.000,C 180.000} C_DIS
LIN {X 61.518,Y 44.779,Z 79.045,A 180.000,B 0.000,C 180.000} C_DIS
LIN {X 61.441,Y 44.796,Z 79.044,A 180.000,B 0.000,C 180.000} C_DIS
LIN {X 61.365,Y 44.816,Z 79.042,A 180.000,B 0.000,C 180.000} C_DIS
LIN {X 61.289,Y 44.838,Z 79.041,A 180.000,B 0.000,C 180.000} C_DIS
LIN {X 61.214,Y 44.862,Z 79.040,A 180.000,B 0.000,C 180.000} C_DIS
LIN {X 61.065,Y 44.912,Z 79.037,A 180.000,B 0.000,C 180.000} C_DIS
LIN {X 60.916,Y 44.963,Z 79.034,A 180.000,B 0.000,C 180.000} C_DIS
LIN {X 60.767,Y 45.013,Z 79.031,A 180.000,B 0.000,C 180.000} C_DIS
LIN {X 60.468,Y 45.114,Z 79.026,A 180.000,B 0.000,C 180.000} C_DIS
LIN {X 60.170,Y 45.214,Z 79.022,A 180.000,B 0.000,C 180.000} C_DIS
LIN {X 59.871,Y 45.315,Z 79.018,A 180.000,B 0.000,C 180.000} C_DIS
LIN {X 59.573,Y 45.416,Z 79.014,A 180.000,B 0.000,C 180.000} C_DIS
LIN {X 59.274,Y 45.517,Z 79.010,A 180.000,B 0.000,C 180.000} C_DIS
LIN {X 58.976,Y 45.617,Z 79.008,A 180.000,B 0.000,C 180.000} C_DIS
LIN {X 58.677,Y 45.718,Z 79.005,A 180.000,B 0.000,C 180.000} C_DIS
LIN {X 58.379,Y 45.819,Z 79.003,A 180.000,B 0.000,C 180.000} C_DIS
LIN {X 58.081,Y 45.919,Z 79.002,A 180.000,B 0.000,C 180.000} C_DIS
LIN {X 57.782,Y 46.020,Z 79.001,A 180.000,B 0.000,C 180.000} C_DIS
LIN {X 57.484,Y 46.121,Z 79.000,A 180.000,B 0.000,C 180.000} C_DIS
LIN {X 57.293,Y 46.185,Z 79.000,A 180.000,B 0.000,C 180.000} C_DIS
; Cutting Move Starts
LIN {X 45.590,Y 50.133,Z 79.000,A 180.000,B 0.000,C 180.000} C_DIS
LIN {X 45.411,Y 50.194,Z 79.000,A 180.000,B 0.000,C 180.000} C_DIS
LIN {X 45.296,Y 50.238,Z 79.000,A 180.000,B 0.000,C 180.000} C_DIS
LIN {X 45.232,Y 50.265,Z 79.000,A 180.000,B 0.000,C 180.000} C_DIS
LIN {X 45.053,Y 50.353,Z 79.000,A 180.000,B 0.000,C 180.000} C_DIS
LIN {X 44.944,Y 50.416,Z 79.000,A 180.000,B 0.000,C 180.000} C_DIS
LIN {X 44.874,Y 50.461,Z 79.000,A 180.000,B 0.000,C 180.000} C_DIS
LIN {X 44.785,Y 50.522,Z 79.000,A 180.000,B 0.000,C 180.000} C_DIS
LIN {X 44.696,Y 50.590,Z 79.000,A 180.000,B 0.000,C 180.000} C_DIS
LIN {X 44.689,Y 50.595,Z 79.000,A 180.000,B 0.000,C 180.000} C_DIS
LIN {X 44.603,Y 50.667,Z 79.000,A 180.000,B 0.000,C 180.000} C_DIS
LIN {X 44.517,Y 50.746,Z 79.000,A 180.000,B 0.000,C 180.000} C_DIS
LIN {X 44.488,Y 50.774,Z 79.000,A 180.000,B 0.000,C 180.000} C_DIS
LIN {X 44.410,Y 50.855,Z 79.000,A 180.000,B 0.000,C 180.000} C_DIS
LIN {X 44.338,Y 50.936,Z 79.000,A 180.000,B 0.000,C 180.000} C_DIS
LIN {X 44.325,Y 50.953,Z 79.000,A 180.000,B 0.000,C 180.000} C_DIS
LIN {X 44.254,Y 51.042,Z 79.000,A 180.000,B 0.000,C 180.000} C_DIS
LIN {X 44.189,Y 51.131,Z 79.000,A 180.000,B 0.000,C 180.000} C_DIS
LIN {X 44.159,Y 51.176,Z 79.000,A 180.000,B 0.000,C 180.000} C_DIS
LIN {X 44.077,Y 51.310,Z 79.000,A 180.000,B 0.000,C 180.000} C_DIS
LIN {X 43.984,Y 51.489,Z 79.000,A 180.000,B 0.000,C 180.000} C_DIS
LIN {X 43.981,Y 51.497,Z 79.000,A 180.000,B 0.000,C 180.000} C_DIS
LIN {X 43.909,Y 51.668,Z 79.000,A 180.000,B 0.000,C 180.000} C_DIS
LIN {X 43.849,Y 51.847,Z 79.000,A 180.000,B 0.000,C 180.000} C_DIS
LIN {X 43.804,Y 52.025,Z 79.000,A 180.000,B 0.000,C 180.000} C_DIS
LIN {X 43.802,Y 52.035,Z 79.000,A 180.000,B 0.000,C 180.000} C_DIS
LIN {X 43.772,Y 52.204,Z 79.000,A 180.000,B 0.000,C 180.000} C_DIS
LIN {X 43.754,Y 52.383,Z 79.000,A 180.000,B 0.000,C 180.000} C_DIS
LIN {X 43.748,Y 52.562,Z 79.000,A 180.000,B 0.000,C 180.000} C_DIS
LIN {X 43.756,Y 52.740,Z 79.000,A 180.000,B 0.000,C 180.000} C_DIS
LIN {X 43.776,Y 52.919,Z 79.000,A 180.000,B 0.000,C 180.000} C_DIS
LIN {X 43.802,Y 53.064,Z 79.000,A 180.000,B 0.000,C 180.000} C_DIS
LIN {X 43.809,Y 53.098,Z 79.000,A 180.000,B 0.000,C 180.000} C_DIS
LIN {X 43.856,Y 53.277,Z 79.000,A 180.000,B 0.000,C 180.000} C_DIS
LIN {X 43.916,Y 53.455,Z 79.000,A 180.000,B 0.000,C 180.000} C_DIS
LIN {X 50.248,Y 72.226,Z 79.000,A 180.000,B 0.000,C 180.000} C_DIS
LIN {X 50.311,Y 72.405,Z 79.000,A 180.000,B 0.000,C 180.000} C_DIS
LIN {X 50.388,Y 72.584,Z 79.000,A 180.000,B 0.000,C 180.000} C_DIS
LIN {X 50.416,Y 72.640,Z 79.000,A 180.000,B 0.000,C 180.000} C_DIS
LIN {X 50.484,Y 72.763,Z 79.000,A 180.000,B 0.000,C 180.000} C_DIS
LIN {X 50.595,Y 72.936,Z 79.000,A 180.000,B 0.000,C 180.000} C_DIS
LIN {X 50.599,Y 72.941,Z 79.000,A 180.000,B 0.000,C 180.000} C_DIS
LIN {X 50.665,Y 73.031,Z 79.000,A 180.000,B 0.000,C 180.000} C_DIS
LIN {X 50.737,Y 73.120,Z 79.000,A 180.000,B 0.000,C 180.000} C_DIS
LIN {X 50.774,Y 73.162,Z 79.000,A 180.000,B 0.000,C 180.000} C_DIS
LIN {X 50.905,Y 73.299,Z 79.000,A 180.000,B 0.000,C 180.000} C_DIS
LIN {X 50.953,Y 73.343,Z 79.000,A 180.000,B 0.000,C 180.000} C_DIS
LIN {X 51.112,Y 73.478,Z 79.000,A 180.000,B 0.000,C 180.000} C_DIS
LIN {X 51.131,Y 73.493,Z 79.000,A 180.000,B 0.000,C 180.000} C_DIS
LIN {X 51.310,Y 73.616,Z 79.000,A 180.000,B 0.000,C 180.000} C_DIS
LIN {X 51.376,Y 73.656,Z 79.000,A 180.000,B 0.000,C 180.000} C_DIS
LIN {X 51.489,Y 73.719,Z 79.000,A 180.000,B 0.000,C 180.000} C_DIS
LIN {X 51.668,Y 73.803,Z 79.000,A 180.000,B 0.000,C 180.000} C_DIS
LIN {X 51.749,Y 73.835,Z 79.000,A 180.000,B 0.000,C 180.000} C_DIS
LIN {X 51.847,Y 73.870,Z 79.000,A 180.000,B 0.000,C 180.000} C_DIS
LIN {X 52.025,Y 73.923,Z 79.000,A 180.000,B 0.000,C 180.000} C_DIS
LIN {X 52.204,Y 73.961,Z 79.000,A 180.000,B 0.000,C 180.000} C_DIS
LIN {X 52.383,Y 73.987,Z 79.000,A 180.000,B 0.000,C 180.000} C_DIS
LIN {X 52.562,Y 73.999,Z 79.000,A 180.000,B 0.000,C 180.000} C_DIS
LIN {X 52.740,Y 73.998,Z 79.000,A 180.000,B 0.000,C 180.000} C_DIS
LIN {X 52.919,Y 73.985,Z 79.000,A 180.000,B 0.000,C 180.000} C_DIS
LIN {X 53.098,Y 73.958,Z 79.000,A 180.000,B 0.000,C 180.000} C_DIS
LIN {X 53.277,Y 73.918,Z 79.000,A 180.000,B 0.000,C 180.000} C_DIS
LIN {X 53.455,Y 73.864,Z 79.000,A 180.000,B 0.000,C 180.000} C_DIS
LIN {X 69.187,Y 68.557,Z 79.000,A 180.000,B 0.000,C 180.000} C_DIS
LIN {X 69.366,Y 68.494,Z 79.000,A 180.000,B 0.000,C 180.000} C_DIS
LIN {X 69.421,Y 68.472,Z 79.000,A 180.000,B 0.000,C 180.000} C_DIS
LIN {X 69.545,Y 68.417,Z 79.000,A 180.000,B 0.000,C 180.000} C_DIS
LIN {X 69.634,Y 68.373,Z 79.000,A 180.000,B 0.000,C 180.000} C_DIS
LIN {X 69.724,Y 68.323,Z 79.000,A 180.000,B 0.000,C 180.000} C_DIS
LIN {X 69.774,Y 68.293,Z 79.000,A 180.000,B 0.000,C 180.000} C_DIS
LIN {X 69.838,Y 68.253,Z 79.000,A 180.000,B 0.000,C 180.000} C_DIS
LIN {X 69.902,Y 68.209,Z 79.000,A 180.000,B 0.000,C 180.000} C_DIS
LIN {X 69.966,Y 68.164,Z 79.000,A 180.000,B 0.000,C 180.000} C_DIS
LIN {X 70.029,Y 68.115,Z 79.000,A 180.000,B 0.000,C 180.000} C_DIS
LIN {X 70.081,Y 68.072,Z 79.000,A 180.000,B 0.000,C 180.000} C_DIS
LIN {X 70.156,Y 68.007,Z 79.000,A 180.000,B 0.000,C 180.000} C_DIS
LIN {X 70.230,Y 67.936,Z 79.000,A 180.000,B 0.000,C 180.000} C_DIS
LIN {X 70.260,Y 67.906,Z 79.000,A 180.000,B 0.000,C 180.000} C_DIS
LIN {X 70.329,Y 67.831,Z 79.000,A 180.000,B 0.000,C 180.000} C_DIS
LIN {X 70.394,Y 67.757,Z 79.000,A 180.000,B 0.000,C 180.000} C_DIS
LIN {X 70.439,Y 67.701,Z 79.000,A 180.000,B 0.000,C 180.000} C_DIS
LIN {X 70.529,Y 67.578,Z 79.000,A 180.000,B 0.000,C 180.000} C_DIS
LIN {X 70.617,Y 67.441,Z 79.000,A 180.000,B 0.000,C 180.000} C_DIS
LIN {X 70.641,Y 67.399,Z 79.000,A 180.000,B 0.000,C 180.000} C_DIS
LIN {X 70.734,Y 67.221,Z 79.000,A 180.000,B 0.000,C 180.000} C_DIS
LIN {X 70.796,Y 67.077,Z 79.000,A 180.000,B 0.000,C 180.000} C_DIS
LIN {X 70.810,Y 67.042,Z 79.000,A 180.000,B 0.000,C 180.000} C_DIS
LIN {X 70.869,Y 66.863,Z 79.000,A 180.000,B 0.000,C 180.000} C_DIS
LIN {X 70.915,Y 66.684,Z 79.000,A 180.000,B 0.000,C 180.000} C_DIS
LIN {X 70.946,Y 66.506,Z 79.000,A 180.000,B 0.000,C 180.000} C_DIS
LIN {X 70.965,Y 66.327,Z 79.000,A 180.000,B 0.000,C 180.000} C_DIS
LIN {X 70.970,Y 66.148,Z 79.000,A 180.000,B 0.000,C 180.000} C_DIS
LIN {X 70.963,Y 65.969,Z 79.000,A 180.000,B 0.000,C 180.000} C_DIS
LIN {X 70.943,Y 65.791,Z 79.000,A 180.000,B 0.000,C 180.000} C_DIS
LIN {X 70.909,Y 65.612,Z 79.000,A 180.000,B 0.000,C 180.000} C_DIS
LIN {X 70.862,Y 65.433,Z 79.000,A 180.000,B 0.000,C 180.000} C_DIS
LIN {X 70.803,Y 65.254,Z 79.000,A 180.000,B 0.000,C 180.000} C_DIS
LIN {X 64.471,Y 46.483,Z 79.000,A 180.000,B 0.000,C 180.000} C_DIS
LIN {X 64.408,Y 46.305,Z 79.000,A 180.000,B 0.000,C 180.000} C_DIS
LIN {X 64.360,Y 46.191,Z 79.000,A 180.000,B 0.000,C 180.000} C_DIS
LIN {X 64.330,Y 46.126,Z 79.000,A 180.000,B 0.000,C 180.000} C_DIS
LIN {X 64.235,Y 45.947,Z 79.000,A 180.000,B 0.000,C 180.000} C_DIS
LIN {X 64.182,Y 45.860,Z 79.000,A 180.000,B 0.000,C 180.000} C_DIS
LIN {X 64.120,Y 45.768,Z 79.000,A 180.000,B 0.000,C 180.000} C_DIS
LIN {X 64.003,Y 45.615,Z 79.000,A 180.000,B 0.000,C 180.000} C_DIS
LIN {X 63.981,Y 45.590,Z 79.000,A 180.000,B 0.000,C 180.000} C_DIS
LIN {X 63.824,Y 45.421,Z 79.000,A 180.000,B 0.000,C 180.000} C_DIS
LIN {X 63.814,Y 45.411,Z 79.000,A 180.000,B 0.000,C 180.000} C_DIS
LIN {X 63.645,Y 45.262,Z 79.000,A 180.000,B 0.000,C 180.000} C_DIS
LIN {X 63.607,Y 45.232,Z 79.000,A 180.000,B 0.000,C 180.000} C_DIS
LIN {X 63.467,Y 45.131,Z 79.000,A 180.000,B 0.000,C 180.000} C_DIS
LIN {X 63.343,Y 45.053,Z 79.000,A 180.000,B 0.000,C 180.000} C_DIS
LIN {X 63.288,Y 45.022,Z 79.000,A 180.000,B 0.000,C 180.000} C_DIS
LIN {X 63.109,Y 44.932,Z 79.000,A 180.000,B 0.000,C 180.000} C_DIS
LIN {X 62.971,Y 44.874,Z 79.000,A 180.000,B 0.000,C 180.000} C_DIS
LIN {X 62.930,Y 44.859,Z 79.000,A 180.000,B 0.000,C 180.000} C_DIS
LIN {X 62.751,Y 44.802,Z 79.000,A 180.000,B 0.000,C 180.000} C_DIS
LIN {X 62.573,Y 44.759,Z 79.000,A 180.000,B 0.000,C 180.000} C_DIS
LIN {X 62.394,Y 44.730,Z 79.000,A 180.000,B 0.000,C 180.000} C_DIS
LIN {X 62.305,Y 44.720,Z 79.000,A 180.000,B 0.000,C 180.000} C_DIS
LIN {X 62.215,Y 44.713,Z 79.000,A 180.000,B 0.000,C 180.000} C_DIS
LIN {X 62.126,Y 44.710,Z 79.000,A 180.000,B 0.000,C 180.000} C_DIS
LIN {X 62.036,Y 44.710,Z 79.000,A 180.000,B 0.000,C 180.000} C_DIS
LIN {X 61.947,Y 44.713,Z 79.000,A 180.000,B 0.000,C 180.000} C_DIS
LIN {X 61.858,Y 44.719,Z 79.000,A 180.000,B 0.000,C 180.000} C_DIS
LIN {X 61.768,Y 44.729,Z 79.000,A 180.000,B 0.000,C 180.000} C_DIS
LIN {X 61.679,Y 44.741,Z 79.000,A 180.000,B 0.000,C 180.000} C_DIS
LIN {X 61.589,Y 44.757,Z 79.000,A 180.000,B 0.000,C 180.000} C_DIS
LIN {X 61.500,Y 44.777,Z 79.000,A 180.000,B 0.000,C 180.000} C_DIS
LIN {X 61.411,Y 44.800,Z 79.000,A 180.000,B 0.000,C 180.000} C_DIS
LIN {X 61.321,Y 44.826,Z 79.000,A 180.000,B 0.000,C 180.000} C_DIS
LIN {X 61.178,Y 44.874,Z 79.000,A 180.000,B 0.000,C 180.000} C_DIS
LIN {X 57.293,Y 46.185,Z 79.000,A 180.000,B 0.000,C 180.000} C_DIS
; Link Move Starts
LIN {X 56.994,Y 46.286,Z 79.000,A 180.000,B 0.000,C 180.000} C_DIS
LIN {X 56.696,Y 46.386,Z 78.999,A 180.000,B 0.000,C 180.000} C_DIS
LIN {X 56.397,Y 46.487,Z 78.998,A 180.000,B 0.000,C 180.000} C_DIS
LIN {X 56.099,Y 46.588,Z 78.996,A 180.000,B 0.000,C 180.000} C_DIS
LIN {X 55.800,Y 46.689,Z 78.994,A 180.000,B 0.000,C 180.000} C_DIS
LIN {X 55.502,Y 46.789,Z 78.991,A 180.000,B 0.000,C 180.000} C_DIS
LIN {X 55.203,Y 46.890,Z 78.988,A 180.000,B 0.000,C 180.000} C_DIS
LIN {X 54.905,Y 46.991,Z 78.985,A 180.000,B 0.000,C 180.000} C_DIS
LIN {X 54.606,Y 47.091,Z 78.981,A 180.000,B 0.000,C 180.000} C_DIS
LIN {X 54.308,Y 47.192,Z 78.977,A 180.000,B 0.000,C 180.000} C_DIS
LIN {X 54.009,Y 47.293,Z 78.972,A 180.000,B 0.000,C 180.000} C_DIS
LIN {X 53.860,Y 47.343,Z 78.969,A 180.000,B 0.000,C 180.000} C_DIS
LIN {X 53.711,Y 47.393,Z 78.967,A 180.000,B 0.000,C 180.000} C_DIS
LIN {X 53.562,Y 47.444,Z 78.964,A 180.000,B 0.000,C 180.000} C_DIS
LIN {X 53.412,Y 47.494,Z 78.961,A 180.000,B 0.000,C 180.000} C_DIS
LIN {X 53.263,Y 47.544,Z 78.959,A 180.000,B 0.000,C 180.000} C_DIS
LIN {X 53.114,Y 47.595,Z 78.956,A 180.000,B 0.000,C 180.000} C_DIS
LIN {X 52.965,Y 47.645,Z 78.952,A 180.000,B 0.000,C 180.000} C_DIS
LIN {X 52.816,Y 47.695,Z 78.949,A 180.000,B 0.000,C 180.000} C_DIS
LIN {X 52.666,Y 47.746,Z 78.946,A 180.000,B 0.000,C 180.000} C_DIS
LIN {X 52.517,Y 47.796,Z 78.943,A 180.000,B 0.000,C 180.000} C_DIS
LIN {X 52.368,Y 47.846,Z 78.939,A 180.000,B 0.000,C 180.000} C_DIS
LIN {X 52.219,Y 47.897,Z 78.936,A 180.000,B 0.000,C 180.000} C_DIS
LIN {X 52.069,Y 47.947,Z 78.932,A 180.000,B 0.000,C 180.000} C_DIS
LIN {X 51.920,Y 47.997,Z 78.928,A 180.000,B 0.000,C 180.000} C_DIS
LIN {X 51.771,Y 48.048,Z 78.925,A 180.000,B 0.000,C 180.000} C_DIS
LIN {X 51.622,Y 48.098,Z 78.921,A 180.000,B 0.000,C 180.000} C_DIS
LIN {X 51.472,Y 48.149,Z 78.917,A 180.000,B 0.000,C 180.000} C_DIS
LIN {X 51.323,Y 48.199,Z 78.913,A 180.000,B 0.000,C 180.000} C_DIS
LIN {X 51.174,Y 48.249,Z 78.909,A 180.000,B 0.000,C 180.000} C_DIS
LIN {X 51.025,Y 48.300,Z 78.905,A 180.000,B 0.000,C 180.000} C_DIS
LIN {X 50.875,Y 48.350,Z 78.900,A 180.000,B 0.000,C 180.000} C_DIS
LIN {X 50.726,Y 48.400,Z 78.896,A 180.000,B 0.000,C 180.000} C_DIS
LIN {X 50.577,Y 48.451,Z 78.892,A 180.000,B 0.000,C 180.000} C_DIS
LIN {X 50.428,Y 48.501,Z 78.887,A 180.000,B 0.000,C 180.000} C_DIS
LIN {X 50.279,Y 48.551,Z 78.883,A 180.000,B 0.000,C 180.000} C_DIS
LIN {X 50.129,Y 48.602,Z 78.878,A 180.000,B 0.000,C 180.000} C_DIS
LIN {X 49.980,Y 48.652,Z 78.873,A 180.000,B 0.000,C 180.000} C_DIS
LIN {X 49.831,Y 48.702,Z 78.869,A 180.000,B 0.000,C 180.000} C_DIS
LIN {X 49.682,Y 48.753,Z 78.864,A 180.000,B 0.000,C 180.000} C_DIS
LIN {X 49.532,Y 48.803,Z 78.859,A 180.000,B 0.000,C 180.000} C_DIS
LIN {X 49.383,Y 48.853,Z 78.854,A 180.000,B 0.000,C 180.000} C_DIS
LIN {X 49.308,Y 48.879,Z 78.851,A 180.000,B 0.000,C 180.000} C_DIS
LIN {X 49.234,Y 48.904,Z 78.849,A 180.000,B 0.000,C 180.000} C_DIS
LIN {X 49.159,Y 48.929,Z 78.846,A 180.000,B 0.000,C 180.000} C_DIS
LIN {X 49.085,Y 48.954,Z 78.844,A 180.000,B 0.000,C 180.000} C_DIS
LIN {X 49.010,Y 48.979,Z 78.841,A 180.000,B 0.000,C 180.000} C_DIS
LIN {X 48.935,Y 49.004,Z 78.839,A 180.000,B 0.000,C 180.000} C_DIS
LIN {X 48.861,Y 49.030,Z 78.836,A 180.000,B 0.000,C 180.000} C_DIS
LIN {X 48.712,Y 49.080,Z 78.831,A 180.000,B 0.000,C 180.000} C_DIS
LIN {X 48.562,Y 49.130,Z 78.825,A 180.000,B 0.000,C 180.000} C_DIS
LIN {X 48.413,Y 49.181,Z 78.820,A 180.000,B 0.000,C 180.000} C_DIS
LIN {X 48.264,Y 49.231,Z 78.815,A 180.000,B 0.000,C 180.000} C_DIS
LIN {X 48.115,Y 49.281,Z 78.809,A 180.000,B 0.000,C 180.000} C_DIS
LIN {X 48.040,Y 49.306,Z 78.807,A 180.000,B 0.000,C 180.000} C_DIS
LIN {X 47.891,Y 49.357,Z 78.801,A 180.000,B 0.000,C 180.000} C_DIS
LIN {X 47.667,Y 49.432,Z 78.793,A 180.000,B 0.000,C 180.000} C_DIS
LIN {X 47.518,Y 49.483,Z 78.787,A 180.000,B 0.000,C 180.000} C_DIS
LIN {X 47.443,Y 49.508,Z 78.785,A 180.000,B 0.000,C 180.000} C_DIS
LIN {X 47.294,Y 49.558,Z 78.779,A 180.000,B 0.000,C 180.000} C_DIS
LIN {X 47.070,Y 49.634,Z 78.771,A 180.000,B 0.000,C 180.000} C_DIS
LIN {X 46.921,Y 49.684,Z 78.765,A 180.000,B 0.000,C 180.000} C_DIS
LIN {X 46.846,Y 49.709,Z 78.763,A 180.000,B 0.000,C 180.000} C_DIS
LIN {X 46.697,Y 49.760,Z 78.757,A 180.000,B 0.000,C 180.000} C_DIS
LIN {X 46.473,Y 49.835,Z 78.749,A 180.000,B 0.000,C 180.000} C_DIS
LIN {X 46.324,Y 49.885,Z 78.743,A 180.000,B 0.000,C 180.000} C_DIS
LIN {X 46.249,Y 49.911,Z 78.741,A 180.000,B 0.000,C 180.000} C_DIS
LIN {X 46.100,Y 49.961,Z 78.735,A 180.000,B 0.000,C 180.000} C_DIS
LIN {X 45.876,Y 50.036,Z 78.727,A 180.000,B 0.000,C 180.000} C_DIS
LIN {X 45.727,Y 50.087,Z 78.721,A 180.000,B 0.000,C 180.000} C_DIS
LIN {X 45.652,Y 50.112,Z 78.719,A 180.000,B 0.000,C 180.000} C_DIS
LIN {X 45.503,Y 50.162,Z 78.713,A 180.000,B 0.000,C 180.000} C_DIS
LIN {X 45.428,Y 50.188,Z 78.710,A 180.000,B 0.000,C 180.000} C_DIS
LIN {X 45.354,Y 50.215,Z 78.708,A 180.000,B 0.000,C 180.000} C_DIS
LIN {X 45.281,Y 50.244,Z 78.705,A 180.000,B 0.000,C 180.000} C_DIS
LIN {X 45.209,Y 50.275,Z 78.702,A 180.000,B 0.000,C 180.000} C_DIS
LIN {X 45.138,Y 50.309,Z 78.699,A 180.000,B 0.000,C 180.000} C_DIS
LIN {X 45.068,Y 50.345,Z 78.697,A 180.000,B 0.000,C 180.000} C_DIS
LIN {X 44.999,Y 50.384,Z 78.694,A 180.000,B 0.000,C 180.000} C_DIS
LIN {X 44.932,Y 50.424,Z 78.691,A 180.000,B 0.000,C 180.000} C_DIS
LIN {X 44.865,Y 50.467,Z 78.688,A 180.000,B 0.000,C 180.000} C_DIS
LIN {X 44.800,Y 50.511,Z 78.686,A 180.000,B 0.000,C 180.000} C_DIS
LIN {X 44.737,Y 50.558,Z 78.683,A 180.000,B 0.000,C 180.000} C_DIS
LIN {X 44.675,Y 50.606,Z 78.680,A 180.000,B 0.000,C 180.000} C_DIS
LIN {X 44.615,Y 50.657,Z 78.677,A 180.000,B 0.000,C 180.000} C_DIS
LIN {X 44.556,Y 50.709,Z 78.675,A 180.000,B 0.000,C 180.000} C_DIS
LIN {X 44.499,Y 50.764,Z 78.672,A 180.000,B 0.000,C 180.000} C_DIS
LIN {X 44.443,Y 50.820,Z 78.669,A 180.000,B 0.000,C 180.000} C_DIS
LIN {X 44.390,Y 50.877,Z 78.666,A 180.000,B 0.000,C 180.000} C_DIS
LIN {X 44.338,Y 50.937,Z 78.664,A 180.000,B 0.000,C 180.000} C_DIS
LIN {X 44.288,Y 50.998,Z 78.661,A 180.000,B 0.000,C 180.000} C_DIS
LIN {X 44.240,Y 51.060,Z 78.658,A 180.000,B 0.000,C 180.000} C_DIS
LIN {X 44.194,Y 51.124,Z 78.655,A 180.000,B 0.000,C 180.000} C_DIS
LIN {X 44.150,Y 51.190,Z 78.653,A 180.000,B 0.000,C 180.000} C_DIS
LIN {X 44.109,Y 51.256,Z 78.650,A 180.000,B 0.000,C 180.000} C_DIS
LIN {X 44.069,Y 51.324,Z 78.647,A 180.000,B 0.000,C 180.000} C_DIS
LIN {X 44.031,Y 51.394,Z 78.644,A 180.000,B 0.000,C 180.000} C_DIS
LIN {X 43.996,Y 51.464,Z 78.642,A 180.000,B 0.000,C 180.000} C_DIS
LIN {X 43.963,Y 51.536,Z 78.639,A 180.000,B 0.000,C 180.000} C_DIS
LIN {X 43.932,Y 51.608,Z 78.636,A 180.000,B 0.000,C 180.000} C_DIS
LIN {X 43.904,Y 51.681,Z 78.633,A 180.000,B 0.000,C 180.000} C_DIS
LIN {X 43.878,Y 51.756,Z 78.631,A 180.000,B 0.000,C 180.000} C_DIS
LIN {X 43.854,Y 51.831,Z 78.628,A 180.000,B 0.000,C 180.000} C_DIS
LIN {X 43.832,Y 51.907,Z 78.625,A 180.000,B 0.000,C 180.000} C_DIS
LIN {X 43.813,Y 51.983,Z 78.622,A 180.000,B 0.000,C 180.000} C_DIS
LIN {X 43.797,Y 52.060,Z 78.620,A 180.000,B 0.000,C 180.000} C_DIS
LIN {X 43.782,Y 52.137,Z 78.617,A 180.000,B 0.000,C 180.000} C_DIS
LIN {X 43.771,Y 52.215,Z 78.614,A 180.000,B 0.000,C 180.000} C_DIS
LIN {X 43.761,Y 52.294,Z 78.611,A 180.000,B 0.000,C 180.000} C_DIS
LIN {X 43.755,Y 52.372,Z 78.609,A 180.000,B 0.000,C 180.000} C_DIS
LIN {X 43.750,Y 52.451,Z 78.606,A 180.000,B 0.000,C 180.000} C_DIS
LIN {X 43.748,Y 52.529,Z 78.603,A 180.000,B 0.000,C 180.000} C_DIS
LIN {X 43.749,Y 52.608,Z 78.600,A 180.000,B 0.000,C 180.000} C_DIS
LIN {X 43.752,Y 52.687,Z 78.598,A 180.000,B 0.000,C 180.000} C_DIS
LIN {X 43.758,Y 52.765,Z 78.595,A 180.000,B 0.000,C 180.000} C_DIS
LIN {X 43.766,Y 52.844,Z 78.592,A 180.000,B 0.000,C 180.000} C_DIS
LIN {X 43.776,Y 52.922,Z 78.589,A 180.000,B 0.000,C 180.000} C_DIS
LIN {X 43.789,Y 53.000,Z 78.587,A 180.000,B 0.000,C 180.000} C_DIS
LIN {X 43.805,Y 53.077,Z 78.584,A 180.000,B 0.000,C 180.000} C_DIS
LIN {X 43.822,Y 53.153,Z 78.581,A 180.000,B 0.000,C 180.000} C_DIS
LIN {X 43.843,Y 53.230,Z 78.578,A 180.000,B 0.000,C 180.000} C_DIS
LIN {X 43.865,Y 53.305,Z 78.576,A 180.000,B 0.000,C 180.000} C_DIS
LIN {X 43.890,Y 53.380,Z 78.573,A 180.000,B 0.000,C 180.000} C_DIS
LIN {X 44.242,Y 54.424,Z 78.534,A 180.000,B 0.000,C 180.000} C_DIS
LIN {X 44.494,Y 55.171,Z 78.507,A 180.000,B 0.000,C 180.000} C_DIS
LIN {X 46.357,Y 60.692,Z 78.303,A 180.000,B 0.000,C 180.000} C_DIS
LIN {X 46.382,Y 60.767,Z 78.301,A 180.000,B 0.000,C 180.000} C_DIS
LIN {X 46.432,Y 60.916,Z 78.295,A 180.000,B 0.000,C 180.000} C_DIS
LIN {X 46.583,Y 61.364,Z 78.279,A 180.000,B 0.000,C 180.000} C_DIS
LIN {X 46.634,Y 61.513,Z 78.273,A 180.000,B 0.000,C 180.000} C_DIS
LIN {X 46.709,Y 61.737,Z 78.265,A 180.000,B 0.000,C 180.000} C_DIS
LIN {X 46.760,Y 61.886,Z 78.259,A 180.000,B 0.000,C 180.000} C_DIS
LIN {X 46.785,Y 61.961,Z 78.257,A 180.000,B 0.000,C 180.000} C_DIS
LIN {X 46.835,Y 62.110,Z 78.251,A 180.000,B 0.000,C 180.000} C_DIS
LIN {X 46.911,Y 62.334,Z 78.243,A 180.000,B 0.000,C 180.000} C_DIS
LIN {X 46.961,Y 62.483,Z 78.237,A 180.000,B 0.000,C 180.000} C_DIS
LIN {X 46.986,Y 62.558,Z 78.235,A 180.000,B 0.000,C 180.000} C_DIS
LIN {X 47.037,Y 62.707,Z 78.229,A 180.000,B 0.000,C 180.000} C_DIS
LIN {X 47.112,Y 62.931,Z 78.221,A 180.000,B 0.000,C 180.000} C_DIS
LIN {X 47.162,Y 63.080,Z 78.215,A 180.000,B 0.000,C 180.000} C_DIS
LIN {X 47.188,Y 63.155,Z 78.213,A 180.000,B 0.000,C 180.000} C_DIS
LIN {X 47.238,Y 63.304,Z 78.207,A 180.000,B 0.000,C 180.000} C_DIS
LIN {X 47.313,Y 63.528,Z 78.199,A 180.000,B 0.000,C 180.000} C_DIS
LIN {X 47.364,Y 63.677,Z 78.193,A 180.000,B 0.000,C 180.000} C_DIS
LIN {X 47.465,Y 63.976,Z 78.182,A 180.000,B 0.000,C 180.000} C_DIS
LIN {X 47.515,Y 64.125,Z 78.177,A 180.000,B 0.000,C 180.000} C_DIS
LIN {X 47.565,Y 64.274,Z 78.172,A 180.000,B 0.000,C 180.000} C_DIS
LIN {X 47.616,Y 64.423,Z 78.166,A 180.000,B 0.000,C 180.000} C_DIS
LIN {X 47.641,Y 64.498,Z 78.164,A 180.000,B 0.000,C 180.000} C_DIS
LIN {X 47.666,Y 64.573,Z 78.161,A 180.000,B 0.000,C 180.000} C_DIS
LIN {X 47.691,Y 64.647,Z 78.159,A 180.000,B 0.000,C 180.000} C_DIS
LIN {X 47.716,Y 64.722,Z 78.156,A 180.000,B 0.000,C 180.000} C_DIS
LIN {X 47.741,Y 64.796,Z 78.154,A 180.000,B 0.000,C 180.000} C_DIS
LIN {X 47.767,Y 64.871,Z 78.151,A 180.000,B 0.000,C 180.000} C_DIS
LIN {X 47.792,Y 64.946,Z 78.149,A 180.000,B 0.000,C 180.000} C_DIS
LIN {X 47.842,Y 65.095,Z 78.144,A 180.000,B 0.000,C 180.000} C_DIS
LIN {X 47.892,Y 65.244,Z 78.139,A 180.000,B 0.000,C 180.000} C_DIS
LIN {X 47.943,Y 65.393,Z 78.134,A 180.000,B 0.000,C 180.000} C_DIS
LIN {X 47.993,Y 65.543,Z 78.129,A 180.000,B 0.000,C 180.000} C_DIS
LIN {X 48.043,Y 65.692,Z 78.124,A 180.000,B 0.000,C 180.000} C_DIS
LIN {X 48.094,Y 65.841,Z 78.120,A 180.000,B 0.000,C 180.000} C_DIS
LIN {X 48.144,Y 65.990,Z 78.115,A 180.000,B 0.000,C 180.000} C_DIS
LIN {X 48.195,Y 66.140,Z 78.111,A 180.000,B 0.000,C 180.000} C_DIS
LIN {X 48.245,Y 66.289,Z 78.106,A 180.000,B 0.000,C 180.000} C_DIS
LIN {X 48.295,Y 66.438,Z 78.102,A 180.000,B 0.000,C 180.000} C_DIS
LIN {X 48.346,Y 66.587,Z 78.097,A 180.000,B 0.000,C 180.000} C_DIS
LIN {X 48.396,Y 66.736,Z 78.093,A 180.000,B 0.000,C 180.000} C_DIS
LIN {X 48.446,Y 66.886,Z 78.089,A 180.000,B 0.000,C 180.000} C_DIS
LIN {X 48.497,Y 67.035,Z 78.085,A 180.000,B 0.000,C 180.000} C_DIS
LIN {X 48.547,Y 67.184,Z 78.081,A 180.000,B 0.000,C 180.000} C_DIS
LIN {X 48.597,Y 67.333,Z 78.077,A 180.000,B 0.000,C 180.000} C_DIS
LIN {X 48.648,Y 67.483,Z 78.073,A 180.000,B 0.000,C 180.000} C_DIS
LIN {X 48.698,Y 67.632,Z 78.070,A 180.000,B 0.000,C 180.000} C_DIS
LIN {X 48.748,Y 67.781,Z 78.066,A 180.000,B 0.000,C 180.000} C_DIS
LIN {X 48.799,Y 67.930,Z 78.062,A 180.000,B 0.000,C 180.000} C_DIS
LIN {X 48.849,Y 68.080,Z 78.059,A 180.000,B 0.000,C 180.000} C_DIS
LIN {X 48.899,Y 68.229,Z 78.056,A 180.000,B 0.000,C 180.000} C_DIS
LIN {X 48.950,Y 68.378,Z 78.052,A 180.000,B 0.000,C 180.000} C_DIS
LIN {X 49.000,Y 68.527,Z 78.049,A 180.000,B 0.000,C 180.000} C_DIS
LIN {X 49.050,Y 68.677,Z 78.046,A 180.000,B 0.000,C 180.000} C_DIS
LIN {X 49.101,Y 68.826,Z 78.043,A 180.000,B 0.000,C 180.000} C_DIS
LIN {X 49.151,Y 68.975,Z 78.040,A 180.000,B 0.000,C 180.000} C_DIS
LIN {X 49.201,Y 69.124,Z 78.037,A 180.000,B 0.000,C 180.000} C_DIS
LIN {X 49.252,Y 69.273,Z 78.034,A 180.000,B 0.000,C 180.000} C_DIS
LIN {X 49.302,Y 69.423,Z 78.032,A 180.000,B 0.000,C 180.000} C_DIS
LIN {X 49.352,Y 69.572,Z 78.029,A 180.000,B 0.000,C 180.000} C_DIS
LIN {X 49.403,Y 69.721,Z 78.027,A 180.000,B 0.000,C 180.000} C_DIS
LIN {X 49.503,Y 70.020,Z 78.022,A 180.000,B 0.000,C 180.000} C_DIS
LIN {X 49.604,Y 70.318,Z 78.018,A 180.000,B 0.000,C 180.000} C_DIS
LIN {X 49.705,Y 70.617,Z 78.014,A 180.000,B 0.000,C 180.000} C_DIS
LIN {X 49.806,Y 70.915,Z 78.011,A 180.000,B 0.000,C 180.000} C_DIS
LIN {X 49.906,Y 71.214,Z 78.008,A 180.000,B 0.000,C 180.000} C_DIS
LIN {X 50.007,Y 71.512,Z 78.005,A 180.000,B 0.000,C 180.000} C_DIS
LIN {X 50.108,Y 71.810,Z 78.003,A 180.000,B 0.000,C 180.000} C_DIS
LIN {X 50.208,Y 72.109,Z 78.002,A 180.000,B 0.000,C 180.000} C_DIS
LIN {X 50.311,Y 72.407,Z 78.001,A 180.000,B 0.000,C 180.000} C_DIS
LIN {X 50.373,Y 72.551,Z 78.000,A 180.000,B 0.000,C 180.000} C_DIS
LIN {X 50.444,Y 72.692,Z 78.000,A 180.000,B 0.000,C 180.000} C_DIS
LIN {X 50.502,Y 72.793,Z 78.000,A 180.000,B 0.000,C 180.000} C_DIS
LIN {X 50.566,Y 72.891,Z 78.000,A 180.000,B 0.000,C 180.000} C_DIS
; Cutting Move Starts
LIN {X 50.595,Y 72.936,Z 78.000,A 180.000,B 0.000,C 180.000} C_DIS
LIN {X 50.599,Y 72.941,Z 78.000,A 180.000,B 0.000,C 180.000} C_DIS
LIN {X 50.665,Y 73.031,Z 78.000,A 180.000,B 0.000,C 180.000} C_DIS
LIN {X 50.737,Y 73.120,Z 78.000,A 180.000,B 0.000,C 180.000} C_DIS
LIN {X 50.774,Y 73.162,Z 78.000,A 180.000,B 0.000,C 180.000} C_DIS
LIN {X 50.905,Y 73.299,Z 78.000,A 180.000,B 0.000,C 180.000} C_DIS
LIN {X 50.953,Y 73.343,Z 78.000,A 180.000,B 0.000,C 180.000} C_DIS
LIN {X 51.112,Y 73.478,Z 78.000,A 180.000,B 0.000,C 180.000} C_DIS
LIN {X 51.131,Y 73.493,Z 78.000,A 180.000,B 0.000,C 180.000} C_DIS
LIN {X 51.310,Y 73.616,Z 78.000,A 180.000,B 0.000,C 180.000} C_DIS
LIN {X 51.376,Y 73.656,Z 78.000,A 180.000,B 0.000,C 180.000} C_DIS
LIN {X 51.489,Y 73.719,Z 78.000,A 180.000,B 0.000,C 180.000} C_DIS
LIN {X 51.668,Y 73.803,Z 78.000,A 180.000,B 0.000,C 180.000} C_DIS
LIN {X 51.749,Y 73.835,Z 78.000,A 180.000,B 0.000,C 180.000} C_DIS
LIN {X 51.847,Y 73.870,Z 78.000,A 180.000,B 0.000,C 180.000} C_DIS
LIN {X 52.025,Y 73.923,Z 78.000,A 180.000,B 0.000,C 180.000} C_DIS
LIN {X 52.204,Y 73.961,Z 78.000,A 180.000,B 0.000,C 180.000} C_DIS
LIN {X 52.383,Y 73.987,Z 78.000,A 180.000,B 0.000,C 180.000} C_DIS
LIN {X 52.562,Y 73.999,Z 78.000,A 180.000,B 0.000,C 180.000} C_DIS
LIN {X 52.740,Y 73.998,Z 78.000,A 180.000,B 0.000,C 180.000} C_DIS
LIN {X 52.919,Y 73.985,Z 78.000,A 180.000,B 0.000,C 180.000} C_DIS
LIN {X 53.098,Y 73.958,Z 78.000,A 180.000,B 0.000,C 180.000} C_DIS
LIN {X 53.277,Y 73.918,Z 78.000,A 180.000,B 0.000,C 180.000} C_DIS
LIN {X 53.455,Y 73.864,Z 78.000,A 180.000,B 0.000,C 180.000} C_DIS
LIN {X 70.260,Y 68.195,Z 78.000,A 180.000,B 0.000,C 180.000} C_DIS
LIN {X 70.439,Y 68.134,Z 78.000,A 180.000,B 0.000,C 180.000} C_DIS
LIN {X 70.493,Y 68.115,Z 78.000,A 180.000,B 0.000,C 180.000} C_DIS
LIN {X 70.617,Y 68.064,Z 78.000,A 180.000,B 0.000,C 180.000} C_DIS
LIN {X 70.707,Y 68.022,Z 78.000,A 180.000,B 0.000,C 180.000} C_DIS
LIN {X 70.796,Y 67.976,Z 78.000,A 180.000,B 0.000,C 180.000} C_DIS
LIN {X 70.868,Y 67.936,Z 78.000,A 180.000,B 0.000,C 180.000} C_DIS
LIN {X 70.975,Y 67.870,Z 78.000,A 180.000,B 0.000,C 180.000} C_DIS
LIN {X 71.054,Y 67.816,Z 78.000,A 180.000,B 0.000,C 180.000} C_DIS
LIN {X 71.134,Y 67.757,Z 78.000,A 180.000,B 0.000,C 180.000} C_DIS
LIN {X 71.154,Y 67.742,Z 78.000,A 180.000,B 0.000,C 180.000} C_DIS
LIN {X 71.243,Y 67.668,Z 78.000,A 180.000,B 0.000,C 180.000} C_DIS
LIN {X 71.332,Y 67.587,Z 78.000,A 180.000,B 0.000,C 180.000} C_DIS
LIN {X 71.342,Y 67.578,Z 78.000,A 180.000,B 0.000,C 180.000} C_DIS
LIN {X 71.430,Y 67.489,Z 78.000,A 180.000,B 0.000,C 180.000} C_DIS
LIN {X 71.510,Y 67.399,Z 78.000,A 180.000,B 0.000,C 180.000} C_DIS
LIN {X 71.511,Y 67.398,Z 78.000,A 180.000,B 0.000,C 180.000} C_DIS
LIN {X 71.583,Y 67.309,Z 78.000,A 180.000,B 0.000,C 180.000} C_DIS
LIN {X 71.649,Y 67.221,Z 78.000,A 180.000,B 0.000,C 180.000} C_DIS
LIN {X 71.690,Y 67.161,Z 78.000,A 180.000,B 0.000,C 180.000} C_DIS
LIN {X 71.765,Y 67.042,Z 78.000,A 180.000,B 0.000,C 180.000} C_DIS
LIN {X 71.860,Y 66.863,Z 78.000,A 180.000,B 0.000,C 180.000} C_DIS
LIN {X 71.869,Y 66.845,Z 78.000,A 180.000,B 0.000,C 180.000} C_DIS
LIN {X 71.938,Y 66.684,Z 78.000,A 180.000,B 0.000,C 180.000} C_DIS
LIN {X 72.000,Y 66.506,Z 78.000,A 180.000,B 0.000,C 180.000} C_DIS
LIN {X 72.048,Y 66.327,Z 78.000,A 180.000,B 0.000,C 180.000} C_DIS
LIN {X 72.048,Y 66.327,Z 78.000,A 180.000,B 0.000,C 180.000} C_DIS
LIN {X 72.081,Y 66.148,Z 78.000,A 180.000,B 0.000,C 180.000} C_DIS
LIN {X 72.102,Y 65.969,Z 78.000,A 180.000,B 0.000,C 180.000} C_DIS
LIN {X 72.109,Y 65.791,Z 78.000,A 180.000,B 0.000,C 180.000} C_DIS
LIN {X 72.104,Y 65.612,Z 78.000,A 180.000,B 0.000,C 180.000} C_DIS
LIN {X 72.085,Y 65.433,Z 78.000,A 180.000,B 0.000,C 180.000} C_DIS
LIN {X 72.054,Y 65.254,Z 78.000,A 180.000,B 0.000,C 180.000} C_DIS
LIN {X 72.048,Y 65.225,Z 78.000,A 180.000,B 0.000,C 180.000} C_DIS
LIN {X 72.009,Y 65.075,Z 78.000,A 180.000,B 0.000,C 180.000} C_DIS
LIN {X 71.951,Y 64.897,Z 78.000,A 180.000,B 0.000,C 180.000} C_DIS
LIN {X 65.612,Y 46.106,Z 78.000,A 180.000,B 0.000,C 180.000} C_DIS
LIN {X 65.557,Y 45.947,Z 78.000,A 180.000,B 0.000,C 180.000} C_DIS
LIN {X 65.482,Y 45.768,Z 78.000,A 180.000,B 0.000,C 180.000} C_DIS
LIN {X 65.433,Y 45.670,Z 78.000,A 180.000,B 0.000,C 180.000} C_DIS
LIN {X 65.389,Y 45.590,Z 78.000,A 180.000,B 0.000,C 180.000} C_DIS
LIN {X 65.277,Y 45.411,Z 78.000,A 180.000,B 0.000,C 180.000} C_DIS
LIN {X 65.254,Y 45.378,Z 78.000,A 180.000,B 0.000,C 180.000} C_DIS
LIN {X 65.143,Y 45.232,Z 78.000,A 180.000,B 0.000,C 180.000} C_DIS
LIN {X 65.075,Y 45.154,Z 78.000,A 180.000,B 0.000,C 180.000} C_DIS
LIN {X 64.980,Y 45.053,Z 78.000,A 180.000,B 0.000,C 180.000} C_DIS
LIN {X 64.897,Y 44.974,Z 78.000,A 180.000,B 0.000,C 180.000} C_DIS
LIN {X 64.780,Y 44.874,Z 78.000,A 180.000,B 0.000,C 180.000} C_DIS
LIN {X 64.718,Y 44.827,Z 78.000,A 180.000,B 0.000,C 180.000} C_DIS
LIN {X 64.539,Y 44.704,Z 78.000,A 180.000,B 0.000,C 180.000} C_DIS
LIN {X 64.526,Y 44.696,Z 78.000,A 180.000,B 0.000,C 180.000} C_DIS
LIN {X 64.360,Y 44.603,Z 78.000,A 180.000,B 0.000,C 180.000} C_DIS
LIN {X 64.182,Y 44.519,Z 78.000,A 180.000,B 0.000,C 180.000} C_DIS
LIN {X 64.176,Y 44.517,Z 78.000,A 180.000,B 0.000,C 180.000} C_DIS
LIN {X 64.003,Y 44.452,Z 78.000,A 180.000,B 0.000,C 180.000} C_DIS
LIN {X 63.824,Y 44.400,Z 78.000,A 180.000,B 0.000,C 180.000} C_DIS
LIN {X 63.645,Y 44.362,Z 78.000,A 180.000,B 0.000,C 180.000} C_DIS
LIN {X 63.470,Y 44.338,Z 78.000,A 180.000,B 0.000,C 180.000} C_DIS
LIN {X 63.467,Y 44.338,Z 78.000,A 180.000,B 0.000,C 180.000} C_DIS
LIN {X 63.377,Y 44.330,Z 78.000,A 180.000,B 0.000,C 180.000} C_DIS
LIN {X 63.288,Y 44.326,Z 78.000,A 180.000,B 0.000,C 180.000} C_DIS
LIN {X 63.198,Y 44.325,Z 78.000,A 180.000,B 0.000,C 180.000} C_DIS
LIN {X 63.109,Y 44.328,Z 78.000,A 180.000,B 0.000,C 180.000} C_DIS
LIN {X 62.962,Y 44.338,Z 78.000,A 180.000,B 0.000,C 180.000} C_DIS
LIN {X 62.930,Y 44.342,Z 78.000,A 180.000,B 0.000,C 180.000} C_DIS
LIN {X 62.841,Y 44.354,Z 78.000,A 180.000,B 0.000,C 180.000} C_DIS
LIN {X 62.751,Y 44.369,Z 78.000,A 180.000,B 0.000,C 180.000} C_DIS
LIN {X 62.662,Y 44.387,Z 78.000,A 180.000,B 0.000,C 180.000} C_DIS
LIN {X 62.573,Y 44.409,Z 78.000,A 180.000,B 0.000,C 180.000} C_DIS
LIN {X 62.483,Y 44.435,Z 78.000,A 180.000,B 0.000,C 180.000} C_DIS
LIN {X 62.394,Y 44.464,Z 78.000,A 180.000,B 0.000,C 180.000} C_DIS
LIN {X 45.590,Y 50.133,Z 78.000,A 180.000,B 0.000,C 180.000} C_DIS
LIN {X 45.411,Y 50.194,Z 78.000,A 180.000,B 0.000,C 180.000} C_DIS
LIN {X 45.296,Y 50.238,Z 78.000,A 180.000,B 0.000,C 180.000} C_DIS
LIN {X 45.232,Y 50.265,Z 78.000,A 180.000,B 0.000,C 180.000} C_DIS
LIN {X 45.053,Y 50.353,Z 78.000,A 180.000,B 0.000,C 180.000} C_DIS
LIN {X 44.944,Y 50.416,Z 78.000,A 180.000,B 0.000,C 180.000} C_DIS
LIN {X 44.874,Y 50.461,Z 78.000,A 180.000,B 0.000,C 180.000} C_DIS
LIN {X 44.785,Y 50.522,Z 78.000,A 180.000,B 0.000,C 180.000} C_DIS
LIN {X 44.696,Y 50.590,Z 78.000,A 180.000,B 0.000,C 180.000} C_DIS
LIN {X 44.689,Y 50.595,Z 78.000,A 180.000,B 0.000,C 180.000} C_DIS
LIN {X 44.603,Y 50.667,Z 78.000,A 180.000,B 0.000,C 180.000} C_DIS
LIN {X 44.517,Y 50.746,Z 78.000,A 180.000,B 0.000,C 180.000} C_DIS
LIN {X 44.488,Y 50.774,Z 78.000,A 180.000,B 0.000,C 180.000} C_DIS
LIN {X 44.410,Y 50.855,Z 78.000,A 180.000,B 0.000,C 180.000} C_DIS
LIN {X 44.338,Y 50.936,Z 78.000,A 180.000,B 0.000,C 180.000} C_DIS
LIN {X 44.325,Y 50.953,Z 78.000,A 180.000,B 0.000,C 180.000} C_DIS
LIN {X 44.254,Y 51.042,Z 78.000,A 180.000,B 0.000,C 180.000} C_DIS
LIN {X 44.189,Y 51.131,Z 78.000,A 180.000,B 0.000,C 180.000} C_DIS
LIN {X 44.159,Y 51.176,Z 78.000,A 180.000,B 0.000,C 180.000} C_DIS
LIN {X 44.077,Y 51.310,Z 78.000,A 180.000,B 0.000,C 180.000} C_DIS
LIN {X 43.984,Y 51.489,Z 78.000,A 180.000,B 0.000,C 180.000} C_DIS
LIN {X 43.981,Y 51.497,Z 78.000,A 180.000,B 0.000,C 180.000} C_DIS
LIN {X 43.909,Y 51.668,Z 78.000,A 180.000,B 0.000,C 180.000} C_DIS
LIN {X 43.849,Y 51.847,Z 78.000,A 180.000,B 0.000,C 180.000} C_DIS
LIN {X 43.804,Y 52.025,Z 78.000,A 180.000,B 0.000,C 180.000} C_DIS
LIN {X 43.802,Y 52.035,Z 78.000,A 180.000,B 0.000,C 180.000} C_DIS
LIN {X 43.772,Y 52.204,Z 78.000,A 180.000,B 0.000,C 180.000} C_DIS
LIN {X 43.754,Y 52.383,Z 78.000,A 180.000,B 0.000,C 180.000} C_DIS
LIN {X 43.748,Y 52.562,Z 78.000,A 180.000,B 0.000,C 180.000} C_DIS
LIN {X 43.756,Y 52.740,Z 78.000,A 180.000,B 0.000,C 180.000} C_DIS
LIN {X 43.776,Y 52.919,Z 78.000,A 180.000,B 0.000,C 180.000} C_DIS
LIN {X 43.802,Y 53.064,Z 78.000,A 180.000,B 0.000,C 180.000} C_DIS
LIN {X 43.809,Y 53.098,Z 78.000,A 180.000,B 0.000,C 180.000} C_DIS
LIN {X 43.856,Y 53.277,Z 78.000,A 180.000,B 0.000,C 180.000} C_DIS
LIN {X 43.916,Y 53.455,Z 78.000,A 180.000,B 0.000,C 180.000} C_DIS
LIN {X 50.248,Y 72.226,Z 78.000,A 180.000,B 0.000,C 180.000} C_DIS
LIN {X 50.311,Y 72.405,Z 78.000,A 180.000,B 0.000,C 180.000} C_DIS
LIN {X 50.388,Y 72.584,Z 78.000,A 180.000,B 0.000,C 180.000} C_DIS
LIN {X 50.416,Y 72.640,Z 78.000,A 180.000,B 0.000,C 180.000} C_DIS
LIN {X 50.484,Y 72.763,Z 78.000,A 180.000,B 0.000,C 180.000} C_DIS
LIN {X 50.566,Y 72.891,Z 78.000,A 180.000,B 0.000,C 180.000} C_DIS
; Link Move Starts
LIN {X 50.656,Y 73.019,Z 78.000,A 180.000,B 0.000,C 180.000} C_DIS
LIN {X 50.756,Y 73.141,Z 78.000,A 180.000,B 0.000,C 180.000} C_DIS
LIN {X 50.863,Y 73.257,Z 77.999,A 180.000,B 0.000,C 180.000} C_DIS
LIN {X 50.977,Y 73.365,Z 77.999,A 180.000,B 0.000,C 180.000} C_DIS
LIN {X 51.098,Y 73.467,Z 77.998,A 180.000,B 0.000,C 180.000} C_DIS
LIN {X 51.225,Y 73.560,Z 77.998,A 180.000,B 0.000,C 180.000} C_DIS
LIN {X 51.357,Y 73.645,Z 77.997,A 180.000,B 0.000,C 180.000} C_DIS
LIN {X 51.495,Y 73.722,Z 77.996,A 180.000,B 0.000,C 180.000} C_DIS
LIN {X 51.637,Y 73.789,Z 77.995,A 180.000,B 0.000,C 180.000} C_DIS
LIN {X 51.783,Y 73.848,Z 77.994,A 180.000,B 0.000,C 180.000} C_DIS
LIN {X 51.933,Y 73.897,Z 77.993,A 180.000,B 0.000,C 180.000} C_DIS
LIN {X 52.085,Y 73.937,Z 77.991,A 180.000,B 0.000,C 180.000} C_DIS
LIN {X 52.240,Y 73.968,Z 77.990,A 180.000,B 0.000,C 180.000} C_DIS
LIN {X 52.396,Y 73.988,Z 77.988,A 180.000,B 0.000,C 180.000} C_DIS
LIN {X 52.553,Y 73.998,Z 77.987,A 180.000,B 0.000,C 180.000} C_DIS
LIN {X 52.710,Y 73.999,Z 77.985,A 180.000,B 0.000,C 180.000} C_DIS
LIN {X 52.868,Y 73.990,Z 77.983,A 180.000,B 0.000,C 180.000} C_DIS
LIN {X 53.024,Y 73.971,Z 77.981,A 180.000,B 0.000,C 180.000} C_DIS
LIN {X 53.179,Y 73.942,Z 77.979,A 180.000,B 0.000,C 180.000} C_DIS
LIN {X 53.331,Y 73.903,Z 77.977,A 180.000,B 0.000,C 180.000} C_DIS
LIN {X 53.631,Y 73.805,Z 77.972,A 180.000,B 0.000,C 180.000} C_DIS
LIN {X 53.780,Y 73.754,Z 77.969,A 180.000,B 0.000,C 180.000} C_DIS
LIN {X 53.929,Y 73.704,Z 77.967,A 180.000,B 0.000,C 180.000} C_DIS
LIN {X 54.078,Y 73.654,Z 77.964,A 180.000,B 0.000,C 180.000} C_DIS
LIN {X 54.228,Y 73.603,Z 77.961,A 180.000,B 0.000,C 180.000} C_DIS
LIN {X 54.377,Y 73.553,Z 77.959,A 180.000,B 0.000,C 180.000} C_DIS
LIN {X 54.526,Y 73.503,Z 77.956,A 180.000,B 0.000,C 180.000} C_DIS
LIN {X 54.675,Y 73.452,Z 77.952,A 180.000,B 0.000,C 180.000} C_DIS
LIN {X 54.825,Y 73.402,Z 77.949,A 180.000,B 0.000,C 180.000} C_DIS
LIN {X 54.974,Y 73.352,Z 77.946,A 180.000,B 0.000,C 180.000} C_DIS
LIN {X 55.123,Y 73.301,Z 77.943,A 180.000,B 0.000,C 180.000} C_DIS
LIN {X 55.272,Y 73.251,Z 77.939,A 180.000,B 0.000,C 180.000} C_DIS
LIN {X 55.422,Y 73.201,Z 77.936,A 180.000,B 0.000,C 180.000} C_DIS
LIN {X 55.571,Y 73.150,Z 77.932,A 180.000,B 0.000,C 180.000} C_DIS
LIN {X 55.720,Y 73.100,Z 77.928,A 180.000,B 0.000,C 180.000} C_DIS
LIN {X 55.869,Y 73.049,Z 77.925,A 180.000,B 0.000,C 180.000} C_DIS
LIN {X 56.019,Y 72.999,Z 77.921,A 180.000,B 0.000,C 180.000} C_DIS
LIN {X 56.168,Y 72.949,Z 77.917,A 180.000,B 0.000,C 180.000} C_DIS
LIN {X 56.317,Y 72.898,Z 77.913,A 180.000,B 0.000,C 180.000} C_DIS
LIN {X 56.466,Y 72.848,Z 77.909,A 180.000,B 0.000,C 180.000} C_DIS
LIN {X 56.615,Y 72.798,Z 77.905,A 180.000,B 0.000,C 180.000} C_DIS
LIN {X 56.765,Y 72.747,Z 77.900,A 180.000,B 0.000,C 180.000} C_DIS
LIN {X 56.914,Y 72.697,Z 77.896,A 180.000,B 0.000,C 180.000} C_DIS
LIN {X 57.063,Y 72.647,Z 77.892,A 180.000,B 0.000,C 180.000} C_DIS
LIN {X 57.212,Y 72.596,Z 77.887,A 180.000,B 0.000,C 180.000} C_DIS
LIN {X 57.362,Y 72.546,Z 77.883,A 180.000,B 0.000,C 180.000} C_DIS
LIN {X 57.511,Y 72.496,Z 77.878,A 180.000,B 0.000,C 180.000} C_DIS
LIN {X 57.660,Y 72.445,Z 77.873,A 180.000,B 0.000,C 180.000} C_DIS
LIN {X 57.809,Y 72.395,Z 77.869,A 180.000,B 0.000,C 180.000} C_DIS
LIN {X 57.959,Y 72.345,Z 77.864,A 180.000,B 0.000,C 180.000} C_DIS
LIN {X 58.108,Y 72.294,Z 77.859,A 180.000,B 0.000,C 180.000} C_DIS
LIN {X 58.257,Y 72.244,Z 77.854,A 180.000,B 0.000,C 180.000} C_DIS
LIN {X 58.332,Y 72.219,Z 77.851,A 180.000,B 0.000,C 180.000} C_DIS
LIN {X 58.406,Y 72.194,Z 77.849,A 180.000,B 0.000,C 180.000} C_DIS
LIN {X 58.481,Y 72.168,Z 77.846,A 180.000,B 0.000,C 180.000} C_DIS
LIN {X 58.556,Y 72.143,Z 77.844,A 180.000,B 0.000,C 180.000} C_DIS
LIN {X 58.630,Y 72.118,Z 77.841,A 180.000,B 0.000,C 180.000} C_DIS
LIN {X 58.705,Y 72.093,Z 77.839,A 180.000,B 0.000,C 180.000} C_DIS
LIN {X 58.779,Y 72.068,Z 77.836,A 180.000,B 0.000,C 180.000} C_DIS
LIN {X 58.929,Y 72.017,Z 77.831,A 180.000,B 0.000,C 180.000} C_DIS
LIN {X 59.078,Y 71.967,Z 77.825,A 180.000,B 0.000,C 180.000} C_DIS
LIN {X 59.227,Y 71.917,Z 77.820,A 180.000,B 0.000,C 180.000} C_DIS
LIN {X 59.376,Y 71.866,Z 77.815,A 180.000,B 0.000,C 180.000} C_DIS
LIN {X 59.526,Y 71.816,Z 77.809,A 180.000,B 0.000,C 180.000} C_DIS
LIN {X 59.600,Y 71.791,Z 77.807,A 180.000,B 0.000,C 180.000} C_DIS
LIN {X 59.749,Y 71.741,Z 77.801,A 180.000,B 0.000,C 180.000} C_DIS
LIN {X 59.973,Y 71.665,Z 77.793,A 180.000,B 0.000,C 180.000} C_DIS
LIN {X 60.123,Y 71.615,Z 77.787,A 180.000,B 0.000,C 180.000} C_DIS
LIN {X 60.197,Y 71.589,Z 77.785,A 180.000,B 0.000,C 180.000} C_DIS
LIN {X 60.346,Y 71.539,Z 77.779,A 180.000,B 0.000,C 180.000} C_DIS
LIN {X 60.570,Y 71.464,Z 77.771,A 180.000,B 0.000,C 180.000} C_DIS
LIN {X 60.719,Y 71.413,Z 77.765,A 180.000,B 0.000,C 180.000} C_DIS
LIN {X 60.794,Y 71.388,Z 77.763,A 180.000,B 0.000,C 180.000} C_DIS
LIN {X 60.943,Y 71.338,Z 77.757,A 180.000,B 0.000,C 180.000} C_DIS
LIN {X 61.167,Y 71.262,Z 77.749,A 180.000,B 0.000,C 180.000} C_DIS
LIN {X 61.316,Y 71.212,Z 77.743,A 180.000,B 0.000,C 180.000} C_DIS
LIN {X 61.391,Y 71.187,Z 77.741,A 180.000,B 0.000,C 180.000} C_DIS
LIN {X 61.540,Y 71.136,Z 77.735,A 180.000,B 0.000,C 180.000} C_DIS
LIN {X 61.764,Y 71.061,Z 77.727,A 180.000,B 0.000,C 180.000} C_DIS
LIN {X 61.913,Y 71.010,Z 77.721,A 180.000,B 0.000,C 180.000} C_DIS
LIN {X 61.988,Y 70.985,Z 77.719,A 180.000,B 0.000,C 180.000} C_DIS
LIN {X 62.137,Y 70.935,Z 77.713,A 180.000,B 0.000,C 180.000} C_DIS
LIN {X 62.585,Y 70.784,Z 77.697,A 180.000,B 0.000,C 180.000} C_DIS
LIN {X 62.734,Y 70.734,Z 77.691,A 180.000,B 0.000,C 180.000} C_DIS
LIN {X 63.182,Y 70.583,Z 77.675,A 180.000,B 0.000,C 180.000} C_DIS
LIN {X 63.331,Y 70.532,Z 77.669,A 180.000,B 0.000,C 180.000} C_DIS
LIN {X 63.853,Y 70.356,Z 77.650,A 180.000,B 0.000,C 180.000} C_DIS
LIN {X 64.301,Y 70.205,Z 77.633,A 180.000,B 0.000,C 180.000} C_DIS
LIN {X 64.450,Y 70.155,Z 77.628,A 180.000,B 0.000,C 180.000} C_DIS
LIN {X 64.898,Y 70.004,Z 77.611,A 180.000,B 0.000,C 180.000} C_DIS
LIN {X 65.047,Y 69.953,Z 77.606,A 180.000,B 0.000,C 180.000} C_DIS
LIN {X 65.794,Y 69.702,Z 77.578,A 180.000,B 0.000,C 180.000} C_DIS
LIN {X 66.167,Y 69.576,Z 77.565,A 180.000,B 0.000,C 180.000} C_DIS
LIN {X 66.614,Y 69.425,Z 77.548,A 180.000,B 0.000,C 180.000} C_DIS
LIN {X 68.331,Y 68.846,Z 77.485,A 180.000,B 0.000,C 180.000} C_DIS
LIN {X 70.868,Y 67.990,Z 77.391,A 180.000,B 0.000,C 180.000} C_DIS
LIN {X 71.091,Y 67.914,Z 77.383,A 180.000,B 0.000,C 180.000} C_DIS
LIN {X 71.166,Y 67.888,Z 77.380,A 180.000,B 0.000,C 180.000} C_DIS
LIN {X 71.239,Y 67.860,Z 77.378,A 180.000,B 0.000,C 180.000} C_DIS
LIN {X 71.312,Y 67.829,Z 77.375,A 180.000,B 0.000,C 180.000} C_DIS
LIN {X 71.384,Y 67.796,Z 77.372,A 180.000,B 0.000,C 180.000} C_DIS
LIN {X 71.455,Y 67.761,Z 77.369,A 180.000,B 0.000,C 180.000} C_DIS
LIN {X 71.526,Y 67.724,Z 77.366,A 180.000,B 0.000,C 180.000} C_DIS
LIN {X 71.593,Y 67.686,Z 77.364,A 180.000,B 0.000,C 180.000} C_DIS
LIN {X 71.660,Y 67.646,Z 77.361,A 180.000,B 0.000,C 180.000} C_DIS
LIN {X 71.725,Y 67.604,Z 77.358,A 180.000,B 0.000,C 180.000} C_DIS
LIN {X 71.789,Y 67.560,Z 77.356,A 180.000,B 0.000,C 180.000} C_DIS
LIN {X 71.851,Y 67.515,Z 77.353,A 180.000,B 0.000,C 180.000} C_DIS
LIN {X 71.911,Y 67.469,Z 77.350,A 180.000,B 0.000,C 180.000} C_DIS
LIN {X 71.970,Y 67.420,Z 77.348,A 180.000,B 0.000,C 180.000} C_DIS
LIN {X 72.027,Y 67.371,Z 77.345,A 180.000,B 0.000,C 180.000} C_DIS
LIN {X 72.082,Y 67.321,Z 77.342,A 180.000,B 0.000,C 180.000} C_DIS
LIN {X 72.135,Y 67.269,Z 77.340,A 180.000,B 0.000,C 180.000} C_DIS
LIN {X 72.187,Y 67.216,Z 77.337,A 180.000,B 0.000,C 180.000} C_DIS
LIN {X 72.238,Y 67.161,Z 77.335,A 180.000,B 0.000,C 180.000} C_DIS
LIN {X 72.287,Y 67.106,Z 77.332,A 180.000,B 0.000,C 180.000} C_DIS
